    TriggL T3459,vl,laserOFF,z0,toolEtna\WObj:=wobjEtna;
    TriggL T3460,v50,laserON,z0,toolEtna\WObj:=wobjEtna;
    TriggL T3461,vl,laserOFF,z0,toolEtna\WObj:=wobjEtna;
    TriggL T3462,v50,laserON,z0,toolEtna\WObj:=wobjEtna;
    TriggL T3463,vl,laserOFF,z0,toolEtna\WObj:=wobjEtna;
    TriggL T3464,v50,laserON,z0,toolEtna\WObj:=wobjEtna;
    TriggL T3465,vl,laserOFF,z0,toolEtna\WObj:=wobjEtna;
    TriggL T3466,v50,laserON,z0,toolEtna\WObj:=wobjEtna;
    TriggL T3467,vl,laserOFF,z0,toolEtna\WObj:=wobjEtna;
    TriggL T3468,v50,laserON,z0,toolEtna\WObj:=wobjEtna;
    TriggL T3469,vl,laserOFF,z0,toolEtna\WObj:=wobjEtna;
    TriggL T3470,v50,laserON,z0,toolEtna\WObj:=wobjEtna;
    TriggL T3471,vl,laserOFF,z0,toolEtna\WObj:=wobjEtna;
    TriggL T3472,v50,laserON,z0,toolEtna\WObj:=wobjEtna;
    TriggL T3473,vl,laserOFF,z0,toolEtna\WObj:=wobjEtna;
    TriggL T3474,v50,laserON,z0,toolEtna\WObj:=wobjEtna;
    TriggL T3475,vl,laserOFF,z0,toolEtna\WObj:=wobjEtna;
    TriggL T3476,v50,laserON,z0,toolEtna\WObj:=wobjEtna;
    TriggL T3477,vl,laserOFF,z0,toolEtna\WObj:=wobjEtna;
    TriggL T3478,v50,laserON,z0,toolEtna\WObj:=wobjEtna;
    TriggL T3479,vl,laserOFF,z0,toolEtna\WObj:=wobjEtna;
    TriggL T3480,v50,laserON,z0,toolEtna\WObj:=wobjEtna;
    TriggL T3481,vl,laserOFF,z0,toolEtna\WObj:=wobjEtna;
    TriggL T3482,v50,laserON,z0,toolEtna\WObj:=wobjEtna;
    TriggL T3483,vl,laserOFF,z0,toolEtna\WObj:=wobjEtna;
    TriggL T3484,v50,laserON,z0,toolEtna\WObj:=wobjEtna;
    TriggL T3485,vl,laserOFF,z0,toolEtna\WObj:=wobjEtna;
    TriggL T3486,v50,laserON,z0,toolEtna\WObj:=wobjEtna;
    TriggL T3487,vl,laserOFF,z0,toolEtna\WObj:=wobjEtna;
    TriggL T3488,v50,laserON,z0,toolEtna\WObj:=wobjEtna;
    TriggL T3489,vl,laserOFF,z0,toolEtna\WObj:=wobjEtna;
    TriggL T3490,v50,laserON,z0,toolEtna\WObj:=wobjEtna;
    TriggL T3491,vl,laserOFF,z0,toolEtna\WObj:=wobjEtna;
    TriggL T3492,v50,laserON,z0,toolEtna\WObj:=wobjEtna;
    TriggL T3493,vl,laserOFF,z0,toolEtna\WObj:=wobjEtna;
    TriggL T3494,v50,laserON,z0,toolEtna\WObj:=wobjEtna;
    TriggL T3495,vl,laserOFF,z0,toolEtna\WObj:=wobjEtna;
    TriggL T3496,v50,laserON,z0,toolEtna\WObj:=wobjEtna;
    TriggL T3497,vl,laserOFF,z0,toolEtna\WObj:=wobjEtna;
    TriggL T3498,v50,laserON,z0,toolEtna\WObj:=wobjEtna;
    TriggL T3499,vl,laserOFF,z0,toolEtna\WObj:=wobjEtna;
    TriggL T3500,v50,laserON,z0,toolEtna\WObj:=wobjEtna;
    TriggL T3501,vl,laserOFF,z0,toolEtna\WObj:=wobjEtna;
    TriggL T3502,v50,laserON,z0,toolEtna\WObj:=wobjEtna;
    TriggL T3503,vl,laserOFF,z0,toolEtna\WObj:=wobjEtna;
    TriggL T3504,v50,laserON,z0,toolEtna\WObj:=wobjEtna;
    TriggL T3505,vl,laserOFF,z0,toolEtna\WObj:=wobjEtna;
    TriggL T3506,v50,laserON,z0,toolEtna\WObj:=wobjEtna;
    TriggL T3507,vl,laserOFF,z0,toolEtna\WObj:=wobjEtna;
    TriggL T3508,v50,laserON,z0,toolEtna\WObj:=wobjEtna;
    TriggL T3509,vl,laserOFF,z0,toolEtna\WObj:=wobjEtna;
    TriggL T3510,v50,laserON,z0,toolEtna\WObj:=wobjEtna;
    TriggL T3511,vl,laserOFF,z0,toolEtna\WObj:=wobjEtna;
    TriggL T3512,v50,laserON,z0,toolEtna\WObj:=wobjEtna;
    TriggL T3513,vl,laserOFF,z0,toolEtna\WObj:=wobjEtna;
    TriggL T3514,v50,laserON,z0,toolEtna\WObj:=wobjEtna;
    TriggL T3515,vl,laserOFF,z0,toolEtna\WObj:=wobjEtna;
    TriggL T3516,v50,laserON,z0,toolEtna\WObj:=wobjEtna;
    TriggL T3517,vl,laserOFF,z0,toolEtna\WObj:=wobjEtna;
    TriggL T3518,v50,laserON,z0,toolEtna\WObj:=wobjEtna;
    TriggL T3519,vl,laserOFF,z0,toolEtna\WObj:=wobjEtna;
    TriggL T3520,v50,laserON,z0,toolEtna\WObj:=wobjEtna;
    TriggL T3521,vl,laserOFF,z0,toolEtna\WObj:=wobjEtna;
    TriggL T3522,v50,laserON,z0,toolEtna\WObj:=wobjEtna;
    TriggL T3523,vl,laserOFF,z0,toolEtna\WObj:=wobjEtna;
    TriggL T3524,v50,laserON,z0,toolEtna\WObj:=wobjEtna;
    TriggL T3525,vl,laserOFF,z0,toolEtna\WObj:=wobjEtna;
    TriggL T3526,v50,laserON,z0,toolEtna\WObj:=wobjEtna;
    TriggL T3527,vl,laserOFF,z0,toolEtna\WObj:=wobjEtna;
    TriggL T3528,v50,laserON,z0,toolEtna\WObj:=wobjEtna;
    TriggL T3529,vl,laserOFF,z0,toolEtna\WObj:=wobjEtna;
    TriggL T3530,v50,laserON,z0,toolEtna\WObj:=wobjEtna;
    TriggL T3531,vl,laserOFF,z0,toolEtna\WObj:=wobjEtna;
    TriggL T3532,v50,laserON,z0,toolEtna\WObj:=wobjEtna;
    TriggL T3533,vl,laserOFF,z0,toolEtna\WObj:=wobjEtna;
    TriggL T3534,v50,laserON,z0,toolEtna\WObj:=wobjEtna;
    TriggL T3535,vl,laserOFF,z0,toolEtna\WObj:=wobjEtna;
    TriggL T3536,v50,laserON,z0,toolEtna\WObj:=wobjEtna;
    TriggL T3537,vl,laserOFF,z0,toolEtna\WObj:=wobjEtna;
    TriggL T3538,v50,laserON,z0,toolEtna\WObj:=wobjEtna;
    TriggL T3539,vl,laserOFF,z0,toolEtna\WObj:=wobjEtna;
    TriggL T3540,v50,laserON,z0,toolEtna\WObj:=wobjEtna;
    TriggL T3541,vl,laserOFF,z0,toolEtna\WObj:=wobjEtna;
    TriggL T3542,v50,laserON,z0,toolEtna\WObj:=wobjEtna;
    TriggL T3543,vl,laserOFF,z0,toolEtna\WObj:=wobjEtna;
    TriggL T3544,v50,laserON,z0,toolEtna\WObj:=wobjEtna;
    TriggL T3545,vl,laserOFF,z0,toolEtna\WObj:=wobjEtna;
    TriggL T3546,v50,laserON,z0,toolEtna\WObj:=wobjEtna;
    TriggL T3547,vl,laserOFF,z0,toolEtna\WObj:=wobjEtna;
    TriggL T3548,v50,laserON,z0,toolEtna\WObj:=wobjEtna;
    TriggL T3549,vl,laserOFF,z0,toolEtna\WObj:=wobjEtna;
    TriggL T3550,v50,laserON,z0,toolEtna\WObj:=wobjEtna;
    TriggL T3551,vl,laserOFF,z0,toolEtna\WObj:=wobjEtna;
    TriggL T3552,v50,laserON,z0,toolEtna\WObj:=wobjEtna;
    TriggL T3553,vl,laserOFF,z0,toolEtna\WObj:=wobjEtna;
    TriggL T3554,v50,laserON,z0,toolEtna\WObj:=wobjEtna;
    TriggL T3555,vl,laserOFF,z0,toolEtna\WObj:=wobjEtna;
    TriggL T3556,v50,laserON,z0,toolEtna\WObj:=wobjEtna;
    TriggL T3557,vl,laserOFF,z0,toolEtna\WObj:=wobjEtna;
    TriggL T3558,v50,laserON,z0,toolEtna\WObj:=wobjEtna;
    TriggL T3559,vl,laserOFF,z0,toolEtna\WObj:=wobjEtna;
    TriggL T3560,v50,laserON,z0,toolEtna\WObj:=wobjEtna;
    TriggL T3561,vl,laserOFF,z0,toolEtna\WObj:=wobjEtna;
    TriggL T3562,v50,laserON,z0,toolEtna\WObj:=wobjEtna;
    TriggL T3563,vl,laserOFF,z0,toolEtna\WObj:=wobjEtna;
    TriggL T3564,v50,laserON,z0,toolEtna\WObj:=wobjEtna;
    TriggL T3565,vl,laserOFF,z0,toolEtna\WObj:=wobjEtna;
    TriggL T3566,v50,laserON,z0,toolEtna\WObj:=wobjEtna;
    TriggL T3567,vl,laserOFF,z0,toolEtna\WObj:=wobjEtna;
    TriggL T3568,v50,laserON,z0,toolEtna\WObj:=wobjEtna;
    TriggL T3569,vl,laserOFF,z0,toolEtna\WObj:=wobjEtna;
    TriggL T3570,v50,laserON,z0,toolEtna\WObj:=wobjEtna;
    TriggL T3571,vl,laserOFF,z0,toolEtna\WObj:=wobjEtna;
    TriggL T3572,v50,laserON,z0,toolEtna\WObj:=wobjEtna;
    TriggL T3573,vl,laserOFF,z0,toolEtna\WObj:=wobjEtna;
    TriggL T3574,v50,laserON,z0,toolEtna\WObj:=wobjEtna;
    TriggL T3575,vl,laserOFF,z0,toolEtna\WObj:=wobjEtna;
    TriggL T3576,v50,laserON,z0,toolEtna\WObj:=wobjEtna;
    TriggL T3577,vl,laserOFF,z0,toolEtna\WObj:=wobjEtna;
    TriggL T3578,v50,laserON,z0,toolEtna\WObj:=wobjEtna;
    TriggL T3579,vl,laserOFF,z0,toolEtna\WObj:=wobjEtna;
    TriggL T3580,v50,laserON,z0,toolEtna\WObj:=wobjEtna;
    TriggL T3581,vl,laserOFF,z0,toolEtna\WObj:=wobjEtna;
    TriggL T3582,v50,laserON,z0,toolEtna\WObj:=wobjEtna;
    TriggL T3583,vl,laserOFF,z0,toolEtna\WObj:=wobjEtna;
    TriggL T3584,v50,laserON,z0,toolEtna\WObj:=wobjEtna;
    TriggL T3585,vl,laserOFF,z0,toolEtna\WObj:=wobjEtna;
    TriggL T3586,v50,laserON,z0,toolEtna\WObj:=wobjEtna;
    TriggL T3587,vl,laserOFF,z0,toolEtna\WObj:=wobjEtna;
    TriggL T3588,v50,laserON,z0,toolEtna\WObj:=wobjEtna;
    TriggL T3589,vl,laserOFF,z0,toolEtna\WObj:=wobjEtna;
    TriggL T3590,v50,laserON,z0,toolEtna\WObj:=wobjEtna;
    TriggL T3591,vl,laserOFF,z0,toolEtna\WObj:=wobjEtna;
    TriggL T3592,v50,laserON,z0,toolEtna\WObj:=wobjEtna;
    TriggL T3593,vl,laserOFF,z0,toolEtna\WObj:=wobjEtna;
    TriggL T3594,v50,laserON,z0,toolEtna\WObj:=wobjEtna;
    TriggL T3595,vl,laserOFF,z0,toolEtna\WObj:=wobjEtna;
    TriggL T3596,v50,laserON,z0,toolEtna\WObj:=wobjEtna;
    TriggL T3597,vl,laserOFF,z0,toolEtna\WObj:=wobjEtna;
    TriggL T3598,v50,laserON,z0,toolEtna\WObj:=wobjEtna;
    TriggL T3599,vl,laserOFF,z0,toolEtna\WObj:=wobjEtna;
    TriggL T3600,v50,laserON,z0,toolEtna\WObj:=wobjEtna;
    TriggL T3601,vl,laserOFF,z0,toolEtna\WObj:=wobjEtna;
    TriggL T3602,v50,laserON,z0,toolEtna\WObj:=wobjEtna;
    TriggL T3603,vl,laserOFF,z0,toolEtna\WObj:=wobjEtna;
    TriggL T3604,v50,laserON,z0,toolEtna\WObj:=wobjEtna;
    TriggL T3605,vl,laserOFF,z0,toolEtna\WObj:=wobjEtna;
    TriggL T3606,v50,laserON,z0,toolEtna\WObj:=wobjEtna;
    TriggL T3607,vl,laserOFF,z0,toolEtna\WObj:=wobjEtna;
    TriggL T3608,v50,laserON,z0,toolEtna\WObj:=wobjEtna;
    TriggL T3609,vl,laserOFF,z0,toolEtna\WObj:=wobjEtna;
    TriggL T3610,v50,laserON,z0,toolEtna\WObj:=wobjEtna;
    TriggL T3611,vl,laserOFF,z0,toolEtna\WObj:=wobjEtna;
    TriggL T3612,v50,laserON,z0,toolEtna\WObj:=wobjEtna;
    TriggL T3613,vl,laserOFF,z0,toolEtna\WObj:=wobjEtna;
    TriggL T3614,v50,laserON,z0,toolEtna\WObj:=wobjEtna;
    TriggL T3615,vl,laserOFF,z0,toolEtna\WObj:=wobjEtna;
    TriggL T3616,v50,laserON,z0,toolEtna\WObj:=wobjEtna;
    TriggL T3617,vl,laserOFF,z0,toolEtna\WObj:=wobjEtna;
    TriggL T3618,v50,laserON,z0,toolEtna\WObj:=wobjEtna;
    TriggL T3619,vl,laserOFF,z0,toolEtna\WObj:=wobjEtna;
    TriggL T3620,v50,laserON,z0,toolEtna\WObj:=wobjEtna;
    TriggL T3621,vl,laserOFF,z0,toolEtna\WObj:=wobjEtna;
    TriggL T3622,v50,laserON,z0,toolEtna\WObj:=wobjEtna;
    TriggL T3623,vl,laserOFF,z0,toolEtna\WObj:=wobjEtna;
    TriggL T3624,v50,laserON,z0,toolEtna\WObj:=wobjEtna;
    TriggL T3625,vl,laserOFF,z0,toolEtna\WObj:=wobjEtna;
    TriggL T3626,v50,laserON,z0,toolEtna\WObj:=wobjEtna;
    TriggL T3627,vl,laserOFF,z0,toolEtna\WObj:=wobjEtna;
    TriggL T3628,v50,laserON,z0,toolEtna\WObj:=wobjEtna;
    TriggL T3629,vl,laserOFF,z0,toolEtna\WObj:=wobjEtna;
    TriggL T3630,v50,laserON,z0,toolEtna\WObj:=wobjEtna;
    TriggL T3631,vl,laserOFF,z0,toolEtna\WObj:=wobjEtna;
    TriggL T3632,v50,laserON,z0,toolEtna\WObj:=wobjEtna;
    TriggL T3633,vl,laserOFF,z0,toolEtna\WObj:=wobjEtna;
    TriggL T3634,v50,laserON,z0,toolEtna\WObj:=wobjEtna;
    TriggL T3635,vl,laserOFF,z0,toolEtna\WObj:=wobjEtna;
    TriggL T3636,v50,laserON,z0,toolEtna\WObj:=wobjEtna;
    TriggL T3637,vl,laserOFF,z0,toolEtna\WObj:=wobjEtna;
    TriggL T3638,v50,laserON,z0,toolEtna\WObj:=wobjEtna;
    TriggL T3639,vl,laserOFF,z0,toolEtna\WObj:=wobjEtna;
    TriggL T3640,v50,laserON,z0,toolEtna\WObj:=wobjEtna;
    TriggL T3641,vl,laserOFF,z0,toolEtna\WObj:=wobjEtna;
    TriggL T3642,v50,laserON,z0,toolEtna\WObj:=wobjEtna;
    TriggL T3643,vl,laserOFF,z0,toolEtna\WObj:=wobjEtna;
    TriggL T3644,v50,laserON,z0,toolEtna\WObj:=wobjEtna;
    TriggL T3645,vl,laserOFF,z0,toolEtna\WObj:=wobjEtna;
    TriggL T3646,v50,laserON,z0,toolEtna\WObj:=wobjEtna;
    TriggL T3647,vl,laserOFF,z0,toolEtna\WObj:=wobjEtna;
    TriggL T3648,v50,laserON,z0,toolEtna\WObj:=wobjEtna;
    TriggL T3649,vl,laserOFF,z0,toolEtna\WObj:=wobjEtna;
    TriggL T3650,v50,laserON,z0,toolEtna\WObj:=wobjEtna;
    TriggL T3651,vl,laserOFF,z0,toolEtna\WObj:=wobjEtna;
    TriggL T3652,v50,laserON,z0,toolEtna\WObj:=wobjEtna;
    TriggL T3653,vl,laserOFF,z0,toolEtna\WObj:=wobjEtna;
    TriggL T3654,v50,laserON,z0,toolEtna\WObj:=wobjEtna;
    TriggL T3655,vl,laserOFF,z0,toolEtna\WObj:=wobjEtna;
    TriggL T3656,v50,laserON,z0,toolEtna\WObj:=wobjEtna;
    TriggL T3657,vl,laserOFF,z0,toolEtna\WObj:=wobjEtna;
    TriggL T3658,v50,laserON,z0,toolEtna\WObj:=wobjEtna;
    TriggL T3659,vl,laserOFF,z0,toolEtna\WObj:=wobjEtna;
    TriggL T3660,v50,laserON,z0,toolEtna\WObj:=wobjEtna;
    TriggL T3661,vl,laserOFF,z0,toolEtna\WObj:=wobjEtna;
    TriggL T3662,v50,laserON,z0,toolEtna\WObj:=wobjEtna;
    TriggL T3663,vl,laserOFF,z0,toolEtna\WObj:=wobjEtna;
    TriggL T3664,v50,laserON,z0,toolEtna\WObj:=wobjEtna;
    TriggL T3665,vl,laserOFF,z0,toolEtna\WObj:=wobjEtna;
    TriggL T3666,v50,laserON,z0,toolEtna\WObj:=wobjEtna;
    TriggL T3667,vl,laserOFF,z0,toolEtna\WObj:=wobjEtna;
    TriggL T3668,v50,laserON,z0,toolEtna\WObj:=wobjEtna;
    TriggL T3669,vl,laserOFF,z0,toolEtna\WObj:=wobjEtna;
    TriggL T3670,v50,laserON,z0,toolEtna\WObj:=wobjEtna;
    TriggL T3671,vl,laserOFF,z0,toolEtna\WObj:=wobjEtna;
    TriggL T3672,v50,laserON,z0,toolEtna\WObj:=wobjEtna;
    TriggL T3673,vl,laserOFF,z0,toolEtna\WObj:=wobjEtna;
    TriggL T3674,v50,laserON,z0,toolEtna\WObj:=wobjEtna;
    TriggL T3675,vl,laserOFF,z0,toolEtna\WObj:=wobjEtna;
    TriggL T3676,v50,laserON,z0,toolEtna\WObj:=wobjEtna;
    TriggL T3677,vl,laserOFF,z0,toolEtna\WObj:=wobjEtna;
    TriggL T3678,v50,laserON,z0,toolEtna\WObj:=wobjEtna;
    TriggL T3679,vl,laserOFF,z0,toolEtna\WObj:=wobjEtna;
    TriggL T3680,v50,laserON,z0,toolEtna\WObj:=wobjEtna;
    TriggL T3681,vl,laserOFF,z0,toolEtna\WObj:=wobjEtna;
    TriggL T3682,v50,laserON,z0,toolEtna\WObj:=wobjEtna;
    TriggL T3683,vl,laserOFF,z0,toolEtna\WObj:=wobjEtna;
    TriggL T3684,v50,laserON,z0,toolEtna\WObj:=wobjEtna;
    TriggL T3685,vl,laserOFF,z0,toolEtna\WObj:=wobjEtna;
    TriggL T3686,v50,laserON,z0,toolEtna\WObj:=wobjEtna;
    TriggL T3687,vl,laserOFF,z0,toolEtna\WObj:=wobjEtna;
    TriggL T3688,v50,laserON,z0,toolEtna\WObj:=wobjEtna;
    TriggL T3689,vl,laserOFF,z0,toolEtna\WObj:=wobjEtna;
    TriggL T3690,v50,laserON,z0,toolEtna\WObj:=wobjEtna;
    TriggL T3691,vl,laserOFF,z0,toolEtna\WObj:=wobjEtna;
    TriggL T3692,v50,laserON,z0,toolEtna\WObj:=wobjEtna;
    TriggL T3693,vl,laserOFF,z0,toolEtna\WObj:=wobjEtna;
    TriggL T3694,v50,laserON,z0,toolEtna\WObj:=wobjEtna;
    TriggL T3695,vl,laserOFF,z0,toolEtna\WObj:=wobjEtna;
    TriggL T3696,v50,laserON,z0,toolEtna\WObj:=wobjEtna;
    TriggL T3697,vl,laserOFF,z0,toolEtna\WObj:=wobjEtna;
    TriggL T3698,v50,laserON,z0,toolEtna\WObj:=wobjEtna;
    TriggL T3699,vl,laserOFF,z0,toolEtna\WObj:=wobjEtna;
    TriggL T3700,v50,laserON,z0,toolEtna\WObj:=wobjEtna;
    TriggL T3701,vl,laserOFF,z0,toolEtna\WObj:=wobjEtna;
    TriggL T3702,v50,laserON,z0,toolEtna\WObj:=wobjEtna;
    TriggL T3703,vl,laserOFF,z0,toolEtna\WObj:=wobjEtna;
    TriggL T3704,v50,laserON,z0,toolEtna\WObj:=wobjEtna;
    TriggL T3705,vl,laserOFF,z0,toolEtna\WObj:=wobjEtna;
    TriggL T3706,v50,laserON,z0,toolEtna\WObj:=wobjEtna;
    TriggL T3707,vl,laserOFF,z0,toolEtna\WObj:=wobjEtna;
    TriggL T3708,v50,laserON,z0,toolEtna\WObj:=wobjEtna;
    TriggL T3709,vl,laserOFF,z0,toolEtna\WObj:=wobjEtna;
    TriggL T3710,v50,laserON,z0,toolEtna\WObj:=wobjEtna;
    TriggL T3711,vl,laserOFF,z0,toolEtna\WObj:=wobjEtna;
    TriggL T3712,v50,laserON,z0,toolEtna\WObj:=wobjEtna;
    TriggL T3713,vl,laserOFF,z0,toolEtna\WObj:=wobjEtna;
    TriggL T3714,v50,laserON,z0,toolEtna\WObj:=wobjEtna;
    TriggL T3715,vl,laserOFF,z0,toolEtna\WObj:=wobjEtna;
    TriggL T3716,v50,laserON,z0,toolEtna\WObj:=wobjEtna;
    TriggL T3717,vl,laserOFF,z0,toolEtna\WObj:=wobjEtna;
    TriggL T3718,v50,laserON,z0,toolEtna\WObj:=wobjEtna;
    TriggL T3719,vl,laserOFF,z0,toolEtna\WObj:=wobjEtna;
    TriggL T3720,v50,laserON,z0,toolEtna\WObj:=wobjEtna;
    TriggL T3721,vl,laserOFF,z0,toolEtna\WObj:=wobjEtna;
    TriggL T3722,v50,laserON,z0,toolEtna\WObj:=wobjEtna;
    TriggL T3723,vl,laserOFF,z0,toolEtna\WObj:=wobjEtna;
    TriggL T3724,v50,laserON,z0,toolEtna\WObj:=wobjEtna;
    TriggL T3725,vl,laserOFF,z0,toolEtna\WObj:=wobjEtna;
    TriggL T3726,v50,laserON,z0,toolEtna\WObj:=wobjEtna;
    TriggL T3727,vl,laserOFF,z0,toolEtna\WObj:=wobjEtna;
    TriggL T3728,v50,laserON,z0,toolEtna\WObj:=wobjEtna;
    TriggL T3729,vl,laserOFF,z0,toolEtna\WObj:=wobjEtna;
    TriggL T3730,v50,laserON,z0,toolEtna\WObj:=wobjEtna;
    TriggL T3731,vl,laserOFF,z0,toolEtna\WObj:=wobjEtna;
    TriggL T3732,v50,laserON,z0,toolEtna\WObj:=wobjEtna;
    TriggL T3733,vl,laserOFF,z0,toolEtna\WObj:=wobjEtna;
    TriggL T3734,v50,laserON,z0,toolEtna\WObj:=wobjEtna;
    TriggL T3735,vl,laserOFF,z0,toolEtna\WObj:=wobjEtna;
    TriggL T3736,v50,laserON,z0,toolEtna\WObj:=wobjEtna;
    TriggL T3737,vl,laserOFF,z0,toolEtna\WObj:=wobjEtna;
    TriggL T3738,v50,laserON,z0,toolEtna\WObj:=wobjEtna;
    TriggL T3739,vl,laserOFF,z0,toolEtna\WObj:=wobjEtna;
    TriggL T3740,v50,laserON,z0,toolEtna\WObj:=wobjEtna;
    TriggL T3741,vl,laserOFF,z0,toolEtna\WObj:=wobjEtna;
    TriggL T3742,v50,laserON,z0,toolEtna\WObj:=wobjEtna;
    TriggL T3743,vl,laserOFF,z0,toolEtna\WObj:=wobjEtna;
    TriggL T3744,v50,laserON,z0,toolEtna\WObj:=wobjEtna;
    TriggL T3745,vl,laserOFF,z0,toolEtna\WObj:=wobjEtna;
    TriggL T3746,v50,laserON,z0,toolEtna\WObj:=wobjEtna;
    TriggL T3747,vl,laserOFF,z0,toolEtna\WObj:=wobjEtna;
    TriggL T3748,v50,laserON,z0,toolEtna\WObj:=wobjEtna;
    TriggL T3749,vl,laserOFF,z0,toolEtna\WObj:=wobjEtna;
    TriggL T3750,v50,laserON,z0,toolEtna\WObj:=wobjEtna;
    TriggL T3751,vl,laserOFF,z0,toolEtna\WObj:=wobjEtna;
    TriggL T3752,v50,laserON,z0,toolEtna\WObj:=wobjEtna;
    TriggL T3753,vl,laserOFF,z0,toolEtna\WObj:=wobjEtna;
    TriggL T3754,v50,laserON,z0,toolEtna\WObj:=wobjEtna;
    TriggL T3755,vl,laserOFF,z0,toolEtna\WObj:=wobjEtna;
    TriggL T3756,v50,laserON,z0,toolEtna\WObj:=wobjEtna;
    TriggL T3757,vl,laserOFF,z0,toolEtna\WObj:=wobjEtna;
    TriggL T3758,v50,laserON,z0,toolEtna\WObj:=wobjEtna;
    TriggL T3759,vl,laserOFF,z0,toolEtna\WObj:=wobjEtna;
    TriggL T3760,v50,laserON,z0,toolEtna\WObj:=wobjEtna;
    TriggL T3761,vl,laserOFF,z0,toolEtna\WObj:=wobjEtna;
    TriggL T3762,v50,laserON,z0,toolEtna\WObj:=wobjEtna;
    TriggL T3763,vl,laserOFF,z0,toolEtna\WObj:=wobjEtna;
    TriggL T3764,v50,laserON,z0,toolEtna\WObj:=wobjEtna;
    TriggL T3765,vl,laserOFF,z0,toolEtna\WObj:=wobjEtna;
    TriggL T3766,v50,laserON,z0,toolEtna\WObj:=wobjEtna;
    TriggL T3767,vl,laserOFF,z0,toolEtna\WObj:=wobjEtna;
    TriggL T3768,v50,laserON,z0,toolEtna\WObj:=wobjEtna;
    TriggL T3769,vl,laserOFF,z0,toolEtna\WObj:=wobjEtna;
    TriggL T3770,v50,laserON,z0,toolEtna\WObj:=wobjEtna;
    TriggL T3771,vl,laserOFF,z0,toolEtna\WObj:=wobjEtna;
    TriggL T3772,v50,laserON,z0,toolEtna\WObj:=wobjEtna;
    TriggL T3773,vl,laserOFF,z0,toolEtna\WObj:=wobjEtna;
    TriggL T3774,v50,laserON,z0,toolEtna\WObj:=wobjEtna;
    TriggL T3775,vl,laserOFF,z0,toolEtna\WObj:=wobjEtna;
    TriggL T3776,v50,laserON,z0,toolEtna\WObj:=wobjEtna;
    TriggL T3777,vl,laserOFF,z0,toolEtna\WObj:=wobjEtna;
    TriggL T3778,v50,laserON,z0,toolEtna\WObj:=wobjEtna;
    TriggL T3779,vl,laserOFF,z0,toolEtna\WObj:=wobjEtna;
    TriggL T3780,v50,laserON,z0,toolEtna\WObj:=wobjEtna;
    TriggL T3781,vl,laserOFF,z0,toolEtna\WObj:=wobjEtna;
    TriggL T3782,v50,laserON,z0,toolEtna\WObj:=wobjEtna;
    TriggL T3783,vl,laserOFF,z0,toolEtna\WObj:=wobjEtna;
    TriggL T3784,v50,laserON,z0,toolEtna\WObj:=wobjEtna;
    TriggL T3785,vl,laserOFF,z0,toolEtna\WObj:=wobjEtna;
    TriggL T3786,v50,laserON,z0,toolEtna\WObj:=wobjEtna;
    TriggL T3787,vl,laserOFF,z0,toolEtna\WObj:=wobjEtna;
    TriggL T3788,v50,laserON,z0,toolEtna\WObj:=wobjEtna;
    TriggL T3789,vl,laserOFF,z0,toolEtna\WObj:=wobjEtna;
    TriggL T3790,v50,laserON,z0,toolEtna\WObj:=wobjEtna;
    TriggL T3791,vl,laserOFF,z0,toolEtna\WObj:=wobjEtna;
    TriggL T3792,v50,laserON,z0,toolEtna\WObj:=wobjEtna;
    TriggL T3793,vl,laserOFF,z0,toolEtna\WObj:=wobjEtna;
    TriggL T3794,v50,laserON,z0,toolEtna\WObj:=wobjEtna;
    TriggL T3795,vl,laserOFF,z0,toolEtna\WObj:=wobjEtna;
    TriggL T3796,v50,laserON,z0,toolEtna\WObj:=wobjEtna;
    TriggL T3797,vl,laserOFF,z0,toolEtna\WObj:=wobjEtna;
    TriggL T3798,v50,laserON,z0,toolEtna\WObj:=wobjEtna;
    TriggL T3799,vl,laserOFF,z0,toolEtna\WObj:=wobjEtna;
    TriggL T3800,v50,laserON,z0,toolEtna\WObj:=wobjEtna;
    TriggL T3801,vl,laserOFF,z0,toolEtna\WObj:=wobjEtna;
    TriggL T3802,v50,laserON,z0,toolEtna\WObj:=wobjEtna;
    TriggL T3803,vl,laserOFF,z0,toolEtna\WObj:=wobjEtna;
    TriggL T3804,v50,laserON,z0,toolEtna\WObj:=wobjEtna;
    TriggL T3805,vl,laserOFF,z0,toolEtna\WObj:=wobjEtna;
    TriggL T3806,v50,laserON,z0,toolEtna\WObj:=wobjEtna;
    TriggL T3807,vl,laserOFF,z0,toolEtna\WObj:=wobjEtna;
    TriggL T3808,v50,laserON,z0,toolEtna\WObj:=wobjEtna;
    TriggL T3809,vl,laserOFF,z0,toolEtna\WObj:=wobjEtna;
    TriggL T3810,v50,laserON,z0,toolEtna\WObj:=wobjEtna;
    TriggL T3811,vl,laserOFF,z0,toolEtna\WObj:=wobjEtna;
    TriggL T3812,v50,laserON,z0,toolEtna\WObj:=wobjEtna;
    TriggL T3813,vl,laserOFF,z0,toolEtna\WObj:=wobjEtna;
    TriggL T3814,v50,laserON,z0,toolEtna\WObj:=wobjEtna;
    TriggL T3815,vl,laserOFF,z0,toolEtna\WObj:=wobjEtna;
    TriggL T3816,v50,laserON,z0,toolEtna\WObj:=wobjEtna;
    TriggL T3817,vl,laserOFF,z0,toolEtna\WObj:=wobjEtna;
    TriggL T3818,v50,laserON,z0,toolEtna\WObj:=wobjEtna;
    TriggL T3819,vl,laserOFF,z0,toolEtna\WObj:=wobjEtna;
    TriggL T3820,v50,laserON,z0,toolEtna\WObj:=wobjEtna;
    TriggL T3821,vl,laserOFF,z0,toolEtna\WObj:=wobjEtna;
    TriggL T3822,v50,laserON,z0,toolEtna\WObj:=wobjEtna;
    TriggL T3823,vl,laserOFF,z0,toolEtna\WObj:=wobjEtna;
    TriggL T3824,v50,laserON,z0,toolEtna\WObj:=wobjEtna;
    TriggL T3825,vl,laserOFF,z0,toolEtna\WObj:=wobjEtna;
    TriggL T3826,v50,laserON,z0,toolEtna\WObj:=wobjEtna;
    TriggL T3827,vl,laserOFF,z0,toolEtna\WObj:=wobjEtna;
    TriggL T3828,v50,laserON,z0,toolEtna\WObj:=wobjEtna;
    TriggL T3829,vl,laserOFF,z0,toolEtna\WObj:=wobjEtna;
    TriggL T3830,v50,laserON,z0,toolEtna\WObj:=wobjEtna;
    TriggL T3831,vl,laserOFF,z0,toolEtna\WObj:=wobjEtna;
    TriggL T3832,v50,laserON,z0,toolEtna\WObj:=wobjEtna;
    TriggL T3833,vl,laserOFF,z0,toolEtna\WObj:=wobjEtna;
    TriggL T3834,v50,laserON,z0,toolEtna\WObj:=wobjEtna;
    TriggL T3835,vl,laserOFF,z0,toolEtna\WObj:=wobjEtna;
    TriggL T3836,v50,laserON,z0,toolEtna\WObj:=wobjEtna;
    TriggL T3837,vl,laserOFF,z0,toolEtna\WObj:=wobjEtna;
    TriggL T3838,v50,laserON,z0,toolEtna\WObj:=wobjEtna;
    TriggL T3839,vl,laserOFF,z0,toolEtna\WObj:=wobjEtna;
    TriggL T3840,v50,laserON,z0,toolEtna\WObj:=wobjEtna;
    TriggL T3841,vl,laserOFF,z0,toolEtna\WObj:=wobjEtna;
    TriggL T3842,v50,laserON,z0,toolEtna\WObj:=wobjEtna;
    TriggL T3843,vl,laserOFF,z0,toolEtna\WObj:=wobjEtna;
    TriggL T3844,v50,laserON,z0,toolEtna\WObj:=wobjEtna;
    TriggL T3845,vl,laserOFF,z0,toolEtna\WObj:=wobjEtna;
    TriggL T3846,v50,laserON,z0,toolEtna\WObj:=wobjEtna;
    TriggL T3847,vl,laserOFF,z0,toolEtna\WObj:=wobjEtna;
    TriggL T3848,v50,laserON,z0,toolEtna\WObj:=wobjEtna;
    TriggL T3849,vl,laserOFF,z0,toolEtna\WObj:=wobjEtna;
    TriggL T3850,v50,laserON,z0,toolEtna\WObj:=wobjEtna;
    TriggL T3851,vl,laserOFF,z0,toolEtna\WObj:=wobjEtna;
    TriggL T3852,v50,laserON,z0,toolEtna\WObj:=wobjEtna;
    TriggL T3853,vl,laserOFF,z0,toolEtna\WObj:=wobjEtna;
    TriggL T3854,v50,laserON,z0,toolEtna\WObj:=wobjEtna;
    TriggL T3855,vl,laserOFF,z0,toolEtna\WObj:=wobjEtna;
    TriggL T3856,v50,laserON,z0,toolEtna\WObj:=wobjEtna;
    TriggL T3857,vl,laserOFF,z0,toolEtna\WObj:=wobjEtna;
    TriggL T3858,v50,laserON,z0,toolEtna\WObj:=wobjEtna;
    TriggL T3859,vl,laserOFF,z0,toolEtna\WObj:=wobjEtna;
    TriggL T3860,v50,laserON,z0,toolEtna\WObj:=wobjEtna;
    TriggL T3861,vl,laserOFF,z0,toolEtna\WObj:=wobjEtna;
    TriggL T3862,v50,laserON,z0,toolEtna\WObj:=wobjEtna;
    TriggL T3863,vl,laserOFF,z0,toolEtna\WObj:=wobjEtna;
    TriggL T3864,v50,laserON,z0,toolEtna\WObj:=wobjEtna;
    TriggL T3865,vl,laserOFF,z0,toolEtna\WObj:=wobjEtna;
    TriggL T3866,v50,laserON,z0,toolEtna\WObj:=wobjEtna;
    TriggL T3867,vl,laserOFF,z0,toolEtna\WObj:=wobjEtna;
    TriggL T3868,v50,laserON,z0,toolEtna\WObj:=wobjEtna;
    TriggL T3869,vl,laserOFF,z0,toolEtna\WObj:=wobjEtna;
    TriggL T3870,v50,laserON,z0,toolEtna\WObj:=wobjEtna;
    TriggL T3871,vl,laserOFF,z0,toolEtna\WObj:=wobjEtna;
    TriggL T3872,v50,laserON,z0,toolEtna\WObj:=wobjEtna;
    TriggL T3873,vl,laserOFF,z0,toolEtna\WObj:=wobjEtna;
    TriggL T3874,v50,laserON,z0,toolEtna\WObj:=wobjEtna;
    TriggL T3875,vl,laserOFF,z0,toolEtna\WObj:=wobjEtna;
    TriggL T3876,v50,laserON,z0,toolEtna\WObj:=wobjEtna;
    TriggL T3877,vl,laserOFF,z0,toolEtna\WObj:=wobjEtna;
    TriggL T3878,v50,laserON,z0,toolEtna\WObj:=wobjEtna;
    TriggL T3879,vl,laserOFF,z0,toolEtna\WObj:=wobjEtna;
    TriggL T3880,v50,laserON,z0,toolEtna\WObj:=wobjEtna;
    TriggL T3881,vl,laserOFF,z0,toolEtna\WObj:=wobjEtna;
    TriggL T3882,v50,laserON,z0,toolEtna\WObj:=wobjEtna;
    TriggL T3883,vl,laserOFF,z0,toolEtna\WObj:=wobjEtna;
    TriggL T3884,v50,laserON,z0,toolEtna\WObj:=wobjEtna;
    TriggL T3885,vl,laserOFF,z0,toolEtna\WObj:=wobjEtna;
    TriggL T3886,v50,laserON,z0,toolEtna\WObj:=wobjEtna;
    TriggL T3887,vl,laserOFF,z0,toolEtna\WObj:=wobjEtna;
    TriggL T3888,v50,laserON,z0,toolEtna\WObj:=wobjEtna;
    TriggL T3889,vl,laserOFF,z0,toolEtna\WObj:=wobjEtna;
    TriggL T3890,v50,laserON,z0,toolEtna\WObj:=wobjEtna;
    TriggL T3891,vl,laserOFF,z0,toolEtna\WObj:=wobjEtna;
    TriggL T3892,v50,laserON,z0,toolEtna\WObj:=wobjEtna;
    TriggL T3893,vl,laserOFF,z0,toolEtna\WObj:=wobjEtna;
    TriggL T3894,v50,laserON,z0,toolEtna\WObj:=wobjEtna;
    TriggL T3895,vl,laserOFF,z0,toolEtna\WObj:=wobjEtna;
    TriggL T3896,v50,laserON,z0,toolEtna\WObj:=wobjEtna;
    TriggL T3897,vl,laserOFF,z0,toolEtna\WObj:=wobjEtna;
    TriggL T3898,v50,laserON,z0,toolEtna\WObj:=wobjEtna;
    TriggL T3899,vl,laserOFF,z0,toolEtna\WObj:=wobjEtna;
    TriggL T3900,v50,laserON,z0,toolEtna\WObj:=wobjEtna;
    TriggL T3901,vl,laserOFF,z0,toolEtna\WObj:=wobjEtna;
    TriggL T3902,v50,laserON,z0,toolEtna\WObj:=wobjEtna;
    TriggL T3903,vl,laserOFF,z0,toolEtna\WObj:=wobjEtna;
    TriggL T3904,v50,laserON,z0,toolEtna\WObj:=wobjEtna;
    TriggL T3905,vl,laserOFF,z0,toolEtna\WObj:=wobjEtna;
    TriggL T3906,v50,laserON,z0,toolEtna\WObj:=wobjEtna;
    TriggL T3907,vl,laserOFF,z0,toolEtna\WObj:=wobjEtna;
    TriggL T3908,v50,laserON,z0,toolEtna\WObj:=wobjEtna;
    TriggL T3909,vl,laserOFF,z0,toolEtna\WObj:=wobjEtna;
    TriggL T3910,v50,laserON,z0,toolEtna\WObj:=wobjEtna;
    TriggL T3911,vl,laserOFF,z0,toolEtna\WObj:=wobjEtna;
    TriggL T3912,v50,laserON,z0,toolEtna\WObj:=wobjEtna;
    TriggL T3913,vl,laserOFF,z0,toolEtna\WObj:=wobjEtna;
    TriggL T3914,v50,laserON,z0,toolEtna\WObj:=wobjEtna;
    TriggL T3915,vl,laserOFF,z0,toolEtna\WObj:=wobjEtna;
    TriggL T3916,v50,laserON,z0,toolEtna\WObj:=wobjEtna;
    TriggL T3917,vl,laserOFF,z0,toolEtna\WObj:=wobjEtna;
    TriggL T3918,v50,laserON,z0,toolEtna\WObj:=wobjEtna;
    TriggL T3919,vl,laserOFF,z0,toolEtna\WObj:=wobjEtna;
    TriggL T3920,v50,laserON,z0,toolEtna\WObj:=wobjEtna;
    TriggL T3921,vl,laserOFF,z0,toolEtna\WObj:=wobjEtna;
    TriggL T3922,v50,laserON,z0,toolEtna\WObj:=wobjEtna;
    TriggL T3923,vl,laserOFF,z0,toolEtna\WObj:=wobjEtna;
    TriggL T3924,v50,laserON,z0,toolEtna\WObj:=wobjEtna;
    TriggL T3925,vl,laserOFF,z0,toolEtna\WObj:=wobjEtna;
    TriggL T3926,v50,laserON,z0,toolEtna\WObj:=wobjEtna;
    TriggL T3927,vl,laserOFF,z0,toolEtna\WObj:=wobjEtna;
    TriggL T3928,v50,laserON,z0,toolEtna\WObj:=wobjEtna;
    TriggL T3929,vl,laserOFF,z0,toolEtna\WObj:=wobjEtna;
    TriggL T3930,v50,laserON,z0,toolEtna\WObj:=wobjEtna;
    TriggL T3931,vl,laserOFF,z0,toolEtna\WObj:=wobjEtna;
    TriggL T3932,v50,laserON,z0,toolEtna\WObj:=wobjEtna;
    TriggL T3933,vl,laserOFF,z0,toolEtna\WObj:=wobjEtna;
    TriggL T3934,v50,laserON,z0,toolEtna\WObj:=wobjEtna;
    TriggL T3935,vl,laserOFF,z0,toolEtna\WObj:=wobjEtna;
    TriggL T3936,v50,laserON,z0,toolEtna\WObj:=wobjEtna;
    TriggL T3937,vl,laserOFF,z0,toolEtna\WObj:=wobjEtna;
    TriggL T3938,v50,laserON,z0,toolEtna\WObj:=wobjEtna;
    TriggL T3939,vl,laserOFF,z0,toolEtna\WObj:=wobjEtna;
    TriggL T3940,v50,laserON,z0,toolEtna\WObj:=wobjEtna;
    TriggL T3941,vl,laserOFF,z0,toolEtna\WObj:=wobjEtna;
    TriggL T3942,v50,laserON,z0,toolEtna\WObj:=wobjEtna;
    TriggL T3943,vl,laserOFF,z0,toolEtna\WObj:=wobjEtna;
    TriggL T3944,v50,laserON,z0,toolEtna\WObj:=wobjEtna;
    TriggL T3945,vl,laserOFF,z0,toolEtna\WObj:=wobjEtna;
    TriggL T3946,v50,laserON,z0,toolEtna\WObj:=wobjEtna;
    TriggL T3947,vl,laserOFF,z0,toolEtna\WObj:=wobjEtna;
    TriggL T3948,v50,laserON,z0,toolEtna\WObj:=wobjEtna;
    TriggL T3949,vl,laserOFF,z0,toolEtna\WObj:=wobjEtna;
    TriggL T3950,v50,laserON,z0,toolEtna\WObj:=wobjEtna;
    TriggL T3951,vl,laserOFF,z0,toolEtna\WObj:=wobjEtna;
    TriggL T3952,v50,laserON,z0,toolEtna\WObj:=wobjEtna;
    TriggL T3953,vl,laserOFF,z0,toolEtna\WObj:=wobjEtna;
    TriggL T3954,v50,laserON,z0,toolEtna\WObj:=wobjEtna;
    TriggL T3955,vl,laserOFF,z0,toolEtna\WObj:=wobjEtna;
    TriggL T3956,v50,laserON,z0,toolEtna\WObj:=wobjEtna;
    TriggL T3957,vl,laserOFF,z0,toolEtna\WObj:=wobjEtna;
    TriggL T3958,v50,laserON,z0,toolEtna\WObj:=wobjEtna;
    TriggL T3959,vl,laserOFF,z0,toolEtna\WObj:=wobjEtna;
    TriggL T3960,v50,laserON,z0,toolEtna\WObj:=wobjEtna;
    TriggL T3961,vl,laserOFF,z0,toolEtna\WObj:=wobjEtna;
    TriggL T3962,v50,laserON,z0,toolEtna\WObj:=wobjEtna;
    TriggL T3963,vl,laserOFF,z0,toolEtna\WObj:=wobjEtna;
    TriggL T3964,v50,laserON,z0,toolEtna\WObj:=wobjEtna;
    TriggL T3965,vl,laserOFF,z0,toolEtna\WObj:=wobjEtna;
    TriggL T3966,v50,laserON,z0,toolEtna\WObj:=wobjEtna;
    TriggL T3967,vl,laserOFF,z0,toolEtna\WObj:=wobjEtna;
    TriggL T3968,v50,laserON,z0,toolEtna\WObj:=wobjEtna;
    TriggL T3969,vl,laserOFF,z0,toolEtna\WObj:=wobjEtna;
    TriggL T3970,v50,laserON,z0,toolEtna\WObj:=wobjEtna;
    TriggL T3971,vl,laserOFF,z0,toolEtna\WObj:=wobjEtna;
    TriggL T3972,v50,laserON,z0,toolEtna\WObj:=wobjEtna;
    TriggL T3973,vl,laserOFF,z0,toolEtna\WObj:=wobjEtna;
    TriggL T3974,v50,laserON,z0,toolEtna\WObj:=wobjEtna;
    TriggL T3975,vl,laserOFF,z0,toolEtna\WObj:=wobjEtna;
    TriggL T3976,v50,laserON,z0,toolEtna\WObj:=wobjEtna;
    TriggL T3977,vl,laserOFF,z0,toolEtna\WObj:=wobjEtna;
    TriggL T3978,v50,laserON,z0,toolEtna\WObj:=wobjEtna;
    TriggL T3979,vl,laserOFF,z0,toolEtna\WObj:=wobjEtna;
    TriggL T3980,v50,laserON,z0,toolEtna\WObj:=wobjEtna;
    TriggL T3981,vl,laserOFF,z0,toolEtna\WObj:=wobjEtna;
    TriggL T3982,v50,laserON,z0,toolEtna\WObj:=wobjEtna;
    TriggL T3983,vl,laserOFF,z0,toolEtna\WObj:=wobjEtna;
    TriggL T3984,v50,laserON,z0,toolEtna\WObj:=wobjEtna;
    TriggL T3985,vl,laserOFF,z0,toolEtna\WObj:=wobjEtna;
    TriggL T3986,v50,laserON,z0,toolEtna\WObj:=wobjEtna;
    TriggL T3987,vl,laserOFF,z0,toolEtna\WObj:=wobjEtna;
    TriggL T3988,v50,laserON,z0,toolEtna\WObj:=wobjEtna;
    TriggL T3989,vl,laserOFF,z0,toolEtna\WObj:=wobjEtna;
    TriggL T3990,v50,laserON,z0,toolEtna\WObj:=wobjEtna;
    TriggL T3991,vl,laserOFF,z0,toolEtna\WObj:=wobjEtna;
    TriggL T3992,v50,laserON,z0,toolEtna\WObj:=wobjEtna;
    TriggL T3993,vl,laserOFF,z0,toolEtna\WObj:=wobjEtna;
    TriggL T3994,v50,laserON,z0,toolEtna\WObj:=wobjEtna;
    TriggL T3995,vl,laserOFF,z0,toolEtna\WObj:=wobjEtna;
    TriggL T3996,v50,laserON,z0,toolEtna\WObj:=wobjEtna;
    TriggL T3997,vl,laserOFF,z0,toolEtna\WObj:=wobjEtna;
    TriggL T3998,v50,laserON,z0,toolEtna\WObj:=wobjEtna;
    TriggL T3999,vl,laserOFF,z0,toolEtna\WObj:=wobjEtna;
    TriggL T4000,v50,laserON,z0,toolEtna\WObj:=wobjEtna;
    TriggL T4001,vl,laserOFF,z0,toolEtna\WObj:=wobjEtna;
    TriggL T4002,v50,laserON,z0,toolEtna\WObj:=wobjEtna;
    TriggL T4003,vl,laserOFF,z0,toolEtna\WObj:=wobjEtna;
    TriggL T4004,v50,laserON,z0,toolEtna\WObj:=wobjEtna;
    TriggL T4005,vl,laserOFF,z0,toolEtna\WObj:=wobjEtna;
    TriggL T4006,v50,laserON,z0,toolEtna\WObj:=wobjEtna;
    TriggL T4007,vl,laserOFF,z0,toolEtna\WObj:=wobjEtna;
    TriggL T4008,v50,laserON,z0,toolEtna\WObj:=wobjEtna;
    TriggL T4009,vl,laserOFF,z0,toolEtna\WObj:=wobjEtna;
    TriggL T4010,v50,laserON,z0,toolEtna\WObj:=wobjEtna;
    TriggL T4011,vl,laserOFF,z0,toolEtna\WObj:=wobjEtna;
    TriggL T4012,v50,laserON,z0,toolEtna\WObj:=wobjEtna;
    TriggL T4013,vl,laserOFF,z0,toolEtna\WObj:=wobjEtna;
    TriggL T4014,v50,laserON,z0,toolEtna\WObj:=wobjEtna;
    TriggL T4015,vl,laserOFF,z0,toolEtna\WObj:=wobjEtna;
    TriggL T4016,v50,laserON,z0,toolEtna\WObj:=wobjEtna;
    TriggL T4017,vl,laserOFF,z0,toolEtna\WObj:=wobjEtna;
    TriggL T4018,v50,laserON,z0,toolEtna\WObj:=wobjEtna;
    TriggL T4019,vl,laserOFF,z0,toolEtna\WObj:=wobjEtna;
    TriggL T4020,v50,laserON,z0,toolEtna\WObj:=wobjEtna;
    TriggL T4021,vl,laserOFF,z0,toolEtna\WObj:=wobjEtna;
    TriggL T4022,v50,laserON,z0,toolEtna\WObj:=wobjEtna;
    TriggL T4023,vl,laserOFF,z0,toolEtna\WObj:=wobjEtna;
    TriggL T4024,v50,laserON,z0,toolEtna\WObj:=wobjEtna;
    TriggL T4025,vl,laserOFF,z0,toolEtna\WObj:=wobjEtna;
    TriggL T4026,v50,laserON,z0,toolEtna\WObj:=wobjEtna;
    TriggL T4027,vl,laserOFF,z0,toolEtna\WObj:=wobjEtna;
    TriggL T4028,v50,laserON,z0,toolEtna\WObj:=wobjEtna;
    TriggL T4029,vl,laserOFF,z0,toolEtna\WObj:=wobjEtna;
    TriggL T4030,v50,laserON,z0,toolEtna\WObj:=wobjEtna;
    TriggL T4031,vl,laserOFF,z0,toolEtna\WObj:=wobjEtna;
    TriggL T4032,v50,laserON,z0,toolEtna\WObj:=wobjEtna;
    TriggL T4033,vl,laserOFF,z0,toolEtna\WObj:=wobjEtna;
    TriggL T4034,v50,laserON,z0,toolEtna\WObj:=wobjEtna;
    TriggL T4035,vl,laserOFF,z0,toolEtna\WObj:=wobjEtna;
    TriggL T4036,v50,laserON,z0,toolEtna\WObj:=wobjEtna;
    TriggL T4037,vl,laserOFF,z0,toolEtna\WObj:=wobjEtna;
    TriggL T4038,v50,laserON,z0,toolEtna\WObj:=wobjEtna;
    TriggL T4039,vl,laserOFF,z0,toolEtna\WObj:=wobjEtna;
    TriggL T4040,v50,laserON,z0,toolEtna\WObj:=wobjEtna;
    TriggL T4041,vl,laserOFF,z0,toolEtna\WObj:=wobjEtna;
    TriggL T4042,v50,laserON,z0,toolEtna\WObj:=wobjEtna;
    TriggL T4043,vl,laserOFF,z0,toolEtna\WObj:=wobjEtna;
    TriggL T4044,v50,laserON,z0,toolEtna\WObj:=wobjEtna;
    TriggL T4045,vl,laserOFF,z0,toolEtna\WObj:=wobjEtna;
    TriggL T4046,v50,laserON,z0,toolEtna\WObj:=wobjEtna;
    TriggL T4047,vl,laserOFF,z0,toolEtna\WObj:=wobjEtna;
    TriggL T4048,v50,laserON,z0,toolEtna\WObj:=wobjEtna;
    TriggL T4049,vl,laserOFF,z0,toolEtna\WObj:=wobjEtna;
    TriggL T4050,v50,laserON,z0,toolEtna\WObj:=wobjEtna;
    TriggL T4051,vl,laserOFF,z0,toolEtna\WObj:=wobjEtna;
    TriggL T4052,v50,laserON,z0,toolEtna\WObj:=wobjEtna;
    TriggL T4053,vl,laserOFF,z0,toolEtna\WObj:=wobjEtna;
    TriggL T4054,v50,laserON,z0,toolEtna\WObj:=wobjEtna;
    TriggL T4055,vl,laserOFF,z0,toolEtna\WObj:=wobjEtna;
    TriggL T4056,v50,laserON,z0,toolEtna\WObj:=wobjEtna;
    TriggL T4057,vl,laserOFF,z0,toolEtna\WObj:=wobjEtna;
    TriggL T4058,v50,laserON,z0,toolEtna\WObj:=wobjEtna;
    TriggL T4059,vl,laserOFF,z0,toolEtna\WObj:=wobjEtna;
    TriggL T4060,v50,laserON,z0,toolEtna\WObj:=wobjEtna;
    TriggL T4061,vl,laserOFF,z0,toolEtna\WObj:=wobjEtna;
    TriggL T4062,v50,laserON,z0,toolEtna\WObj:=wobjEtna;
    TriggL T4063,vl,laserOFF,z0,toolEtna\WObj:=wobjEtna;
    TriggL T4064,v50,laserON,z0,toolEtna\WObj:=wobjEtna;
    TriggL T4065,vl,laserOFF,z0,toolEtna\WObj:=wobjEtna;
    TriggL T4066,v50,laserON,z0,toolEtna\WObj:=wobjEtna;
    TriggL T4067,vl,laserOFF,z0,toolEtna\WObj:=wobjEtna;
    TriggL T4068,v50,laserON,z0,toolEtna\WObj:=wobjEtna;
    TriggL T4069,vl,laserOFF,z0,toolEtna\WObj:=wobjEtna;
    TriggL T4070,v50,laserON,z0,toolEtna\WObj:=wobjEtna;
    TriggL T4071,vl,laserOFF,z0,toolEtna\WObj:=wobjEtna;
    TriggL T4072,v50,laserON,z0,toolEtna\WObj:=wobjEtna;
    TriggL T4073,vl,laserOFF,z0,toolEtna\WObj:=wobjEtna;
    TriggL T4074,v50,laserON,z0,toolEtna\WObj:=wobjEtna;
    TriggL T4075,vl,laserOFF,z0,toolEtna\WObj:=wobjEtna;
    TriggL T4076,v50,laserON,z0,toolEtna\WObj:=wobjEtna;
    TriggL T4077,vl,laserOFF,z0,toolEtna\WObj:=wobjEtna;
    TriggL T4078,v50,laserON,z0,toolEtna\WObj:=wobjEtna;
    TriggL T4079,vl,laserOFF,z0,toolEtna\WObj:=wobjEtna;
    TriggL T4080,v50,laserON,z0,toolEtna\WObj:=wobjEtna;
    TriggL T4081,vl,laserOFF,z0,toolEtna\WObj:=wobjEtna;
    TriggL T4082,v50,laserON,z0,toolEtna\WObj:=wobjEtna;
    TriggL T4083,vl,laserOFF,z0,toolEtna\WObj:=wobjEtna;
    TriggL T4084,v50,laserON,z0,toolEtna\WObj:=wobjEtna;
    TriggL T4085,vl,laserOFF,z0,toolEtna\WObj:=wobjEtna;
    TriggL T4086,v50,laserON,z0,toolEtna\WObj:=wobjEtna;
    TriggL T4087,vl,laserOFF,z0,toolEtna\WObj:=wobjEtna;
    TriggL T4088,v50,laserON,z0,toolEtna\WObj:=wobjEtna;
    TriggL T4089,vl,laserOFF,z0,toolEtna\WObj:=wobjEtna;
    TriggL T4090,v50,laserON,z0,toolEtna\WObj:=wobjEtna;
    TriggL T4091,vl,laserOFF,z0,toolEtna\WObj:=wobjEtna;
    TriggL T4092,v50,laserON,z0,toolEtna\WObj:=wobjEtna;
    TriggL T4093,vl,laserOFF,z0,toolEtna\WObj:=wobjEtna;
    TriggL T4094,v50,laserON,z0,toolEtna\WObj:=wobjEtna;
    TriggL T4095,vl,laserOFF,z0,toolEtna\WObj:=wobjEtna;
    TriggL T4096,v50,laserON,z0,toolEtna\WObj:=wobjEtna;
    TriggL T4097,vl,laserOFF,z0,toolEtna\WObj:=wobjEtna;
    TriggL T4098,v50,laserON,z0,toolEtna\WObj:=wobjEtna;
    TriggL T4099,vl,laserOFF,z0,toolEtna\WObj:=wobjEtna;
    TriggL T4100,v50,laserON,z0,toolEtna\WObj:=wobjEtna;
    TriggL T4101,vl,laserOFF,z0,toolEtna\WObj:=wobjEtna;
    TriggL T4102,v50,laserON,z0,toolEtna\WObj:=wobjEtna;
    TriggL T4103,vl,laserOFF,z0,toolEtna\WObj:=wobjEtna;
    TriggL T4104,v50,laserON,z0,toolEtna\WObj:=wobjEtna;
    TriggL T4105,vl,laserOFF,z0,toolEtna\WObj:=wobjEtna;
    TriggL T4106,v50,laserON,z0,toolEtna\WObj:=wobjEtna;
    TriggL T4107,vl,laserOFF,z0,toolEtna\WObj:=wobjEtna;
    TriggL T4108,v50,laserON,z0,toolEtna\WObj:=wobjEtna;
    TriggL T4109,vl,laserOFF,z0,toolEtna\WObj:=wobjEtna;
    TriggL T4110,v50,laserON,z0,toolEtna\WObj:=wobjEtna;
    TriggL T4111,vl,laserOFF,z0,toolEtna\WObj:=wobjEtna;
    TriggL T4112,v50,laserON,z0,toolEtna\WObj:=wobjEtna;
    TriggL T4113,vl,laserOFF,z0,toolEtna\WObj:=wobjEtna;
    TriggL T4114,v50,laserON,z0,toolEtna\WObj:=wobjEtna;
    TriggL T4115,vl,laserOFF,z0,toolEtna\WObj:=wobjEtna;
    TriggL T4116,v50,laserON,z0,toolEtna\WObj:=wobjEtna;
    TriggL T4117,vl,laserOFF,z0,toolEtna\WObj:=wobjEtna;
    TriggL T4118,v50,laserON,z0,toolEtna\WObj:=wobjEtna;
    TriggL T4119,vl,laserOFF,z0,toolEtna\WObj:=wobjEtna;
    TriggL T4120,v50,laserON,z0,toolEtna\WObj:=wobjEtna;
    TriggL T4121,vl,laserOFF,z0,toolEtna\WObj:=wobjEtna;
    TriggL T4122,v50,laserON,z0,toolEtna\WObj:=wobjEtna;
    TriggL T4123,vl,laserOFF,z0,toolEtna\WObj:=wobjEtna;
    TriggL T4124,v50,laserON,z0,toolEtna\WObj:=wobjEtna;
    TriggL T4125,vl,laserOFF,z0,toolEtna\WObj:=wobjEtna;
    TriggL T4126,v50,laserON,z0,toolEtna\WObj:=wobjEtna;
    TriggL T4127,vl,laserOFF,z0,toolEtna\WObj:=wobjEtna;
    TriggL T4128,v50,laserON,z0,toolEtna\WObj:=wobjEtna;
    TriggL T4129,vl,laserOFF,z0,toolEtna\WObj:=wobjEtna;
    TriggL T4130,v50,laserON,z0,toolEtna\WObj:=wobjEtna;
    TriggL T4131,vl,laserOFF,z0,toolEtna\WObj:=wobjEtna;
    TriggL T4132,v50,laserON,z0,toolEtna\WObj:=wobjEtna;
    TriggL T4133,vl,laserOFF,z0,toolEtna\WObj:=wobjEtna;
    TriggL T4134,v50,laserON,z0,toolEtna\WObj:=wobjEtna;
    TriggL T4135,vl,laserOFF,z0,toolEtna\WObj:=wobjEtna;
    TriggL T4136,v50,laserON,z0,toolEtna\WObj:=wobjEtna;
    TriggL T4137,vl,laserOFF,z0,toolEtna\WObj:=wobjEtna;
    TriggL T4138,v50,laserON,z0,toolEtna\WObj:=wobjEtna;
    TriggL T4139,vl,laserOFF,z0,toolEtna\WObj:=wobjEtna;
    TriggL T4140,v50,laserON,z0,toolEtna\WObj:=wobjEtna;
    TriggL T4141,vl,laserOFF,z0,toolEtna\WObj:=wobjEtna;
    TriggL T4142,v50,laserON,z0,toolEtna\WObj:=wobjEtna;
    TriggL T4143,vl,laserOFF,z0,toolEtna\WObj:=wobjEtna;
    TriggL T4144,v50,laserON,z0,toolEtna\WObj:=wobjEtna;
    TriggL T4145,vl,laserOFF,z0,toolEtna\WObj:=wobjEtna;
    TriggL T4146,v50,laserON,z0,toolEtna\WObj:=wobjEtna;
    TriggL T4147,vl,laserOFF,z0,toolEtna\WObj:=wobjEtna;
    TriggL T4148,v50,laserON,z0,toolEtna\WObj:=wobjEtna;
    TriggL T4149,vl,laserOFF,z0,toolEtna\WObj:=wobjEtna;
    TriggL T4150,v50,laserON,z0,toolEtna\WObj:=wobjEtna;
    TriggL T4151,vl,laserOFF,z0,toolEtna\WObj:=wobjEtna;
    TriggL T4152,v50,laserON,z0,toolEtna\WObj:=wobjEtna;
    TriggL T4153,vl,laserOFF,z0,toolEtna\WObj:=wobjEtna;
    TriggL T4154,v50,laserON,z0,toolEtna\WObj:=wobjEtna;
    TriggL T4155,vl,laserOFF,z0,toolEtna\WObj:=wobjEtna;
    TriggL T4156,v50,laserON,z0,toolEtna\WObj:=wobjEtna;
    TriggL T4157,vl,laserOFF,z0,toolEtna\WObj:=wobjEtna;
    TriggL T4158,v50,laserON,z0,toolEtna\WObj:=wobjEtna;
    TriggL T4159,vl,laserOFF,z0,toolEtna\WObj:=wobjEtna;
    TriggL T4160,v50,laserON,z0,toolEtna\WObj:=wobjEtna;
    TriggL T4161,vl,laserOFF,z0,toolEtna\WObj:=wobjEtna;
    TriggL T4162,v50,laserON,z0,toolEtna\WObj:=wobjEtna;
    TriggL T4163,vl,laserOFF,z0,toolEtna\WObj:=wobjEtna;
    TriggL T4164,v50,laserON,z0,toolEtna\WObj:=wobjEtna;
    TriggL T4165,vl,laserOFF,z0,toolEtna\WObj:=wobjEtna;
    TriggL T4166,v50,laserON,z0,toolEtna\WObj:=wobjEtna;
    TriggL T4167,vl,laserOFF,z0,toolEtna\WObj:=wobjEtna;
    TriggL T4168,v50,laserON,z0,toolEtna\WObj:=wobjEtna;
    TriggL T4169,vl,laserOFF,z0,toolEtna\WObj:=wobjEtna;
    TriggL T4170,v50,laserON,z0,toolEtna\WObj:=wobjEtna;
    TriggL T4171,vl,laserOFF,z0,toolEtna\WObj:=wobjEtna;
    TriggL T4172,v50,laserON,z0,toolEtna\WObj:=wobjEtna;
    TriggL T4173,vl,laserOFF,z0,toolEtna\WObj:=wobjEtna;
    TriggL T4174,v50,laserON,z0,toolEtna\WObj:=wobjEtna;
    TriggL T4175,vl,laserOFF,z0,toolEtna\WObj:=wobjEtna;
    TriggL T4176,v50,laserON,z0,toolEtna\WObj:=wobjEtna;
    TriggL T4177,vl,laserOFF,z0,toolEtna\WObj:=wobjEtna;
    TriggL T4178,v50,laserON,z0,toolEtna\WObj:=wobjEtna;
    TriggL T4179,vl,laserOFF,z0,toolEtna\WObj:=wobjEtna;
    TriggL T4180,v50,laserON,z0,toolEtna\WObj:=wobjEtna;
    TriggL T4181,vl,laserOFF,z0,toolEtna\WObj:=wobjEtna;
    TriggL T4182,v50,laserON,z0,toolEtna\WObj:=wobjEtna;
    TriggL T4183,vl,laserOFF,z0,toolEtna\WObj:=wobjEtna;
    TriggL T4184,v50,laserON,z0,toolEtna\WObj:=wobjEtna;
    TriggL T4185,vl,laserOFF,z0,toolEtna\WObj:=wobjEtna;
    TriggL T4186,v50,laserON,z0,toolEtna\WObj:=wobjEtna;
    TriggL T4187,vl,laserOFF,z0,toolEtna\WObj:=wobjEtna;
    TriggL T4188,v50,laserON,z0,toolEtna\WObj:=wobjEtna;
    TriggL T4189,vl,laserOFF,z0,toolEtna\WObj:=wobjEtna;
    TriggL T4190,v50,laserON,z0,toolEtna\WObj:=wobjEtna;
    TriggL T4191,vl,laserOFF,z0,toolEtna\WObj:=wobjEtna;
    TriggL T4192,v50,laserON,z0,toolEtna\WObj:=wobjEtna;
    TriggL T4193,vl,laserOFF,z0,toolEtna\WObj:=wobjEtna;
    TriggL T4194,v50,laserON,z0,toolEtna\WObj:=wobjEtna;
    TriggL T4195,vl,laserOFF,z0,toolEtna\WObj:=wobjEtna;
    TriggL T4196,v50,laserON,z0,toolEtna\WObj:=wobjEtna;
    TriggL T4197,vl,laserOFF,z0,toolEtna\WObj:=wobjEtna;
    TriggL T4198,v50,laserON,z0,toolEtna\WObj:=wobjEtna;
    TriggL T4199,vl,laserOFF,z0,toolEtna\WObj:=wobjEtna;
    TriggL T4200,v50,laserON,z0,toolEtna\WObj:=wobjEtna;
    TriggL T4201,vl,laserOFF,z0,toolEtna\WObj:=wobjEtna;
    TriggL T4202,v50,laserON,z0,toolEtna\WObj:=wobjEtna;
    TriggL T4203,vl,laserOFF,z0,toolEtna\WObj:=wobjEtna;
    TriggL T4204,v50,laserON,z0,toolEtna\WObj:=wobjEtna;
    TriggL T4205,vl,laserOFF,z0,toolEtna\WObj:=wobjEtna;
    TriggL T4206,v50,laserON,z0,toolEtna\WObj:=wobjEtna;
    TriggL T4207,vl,laserOFF,z0,toolEtna\WObj:=wobjEtna;
    TriggL T4208,v50,laserON,z0,toolEtna\WObj:=wobjEtna;
    TriggL T4209,vl,laserOFF,z0,toolEtna\WObj:=wobjEtna;
    TriggL T4210,v50,laserON,z0,toolEtna\WObj:=wobjEtna;
    TriggL T4211,vl,laserOFF,z0,toolEtna\WObj:=wobjEtna;
    TriggL T4212,v50,laserON,z0,toolEtna\WObj:=wobjEtna;
    TriggL T4213,vl,laserOFF,z0,toolEtna\WObj:=wobjEtna;
    TriggL T4214,v50,laserON,z0,toolEtna\WObj:=wobjEtna;
    TriggL T4215,vl,laserOFF,z0,toolEtna\WObj:=wobjEtna;
    TriggL T4216,v50,laserON,z0,toolEtna\WObj:=wobjEtna;
    TriggL T4217,vl,laserOFF,z0,toolEtna\WObj:=wobjEtna;
    TriggL T4218,v50,laserON,z0,toolEtna\WObj:=wobjEtna;
    TriggL T4219,vl,laserOFF,z0,toolEtna\WObj:=wobjEtna;
    TriggL T4220,v50,laserON,z0,toolEtna\WObj:=wobjEtna;
    TriggL T4221,vl,laserOFF,z0,toolEtna\WObj:=wobjEtna;
    TriggL T4222,v50,laserON,z0,toolEtna\WObj:=wobjEtna;
    TriggL T4223,vl,laserOFF,z0,toolEtna\WObj:=wobjEtna;
    TriggL T4224,v50,laserON,z0,toolEtna\WObj:=wobjEtna;
    TriggL T4225,vl,laserOFF,z0,toolEtna\WObj:=wobjEtna;
    TriggL T4226,v50,laserON,z0,toolEtna\WObj:=wobjEtna;
    TriggL T4227,vl,laserOFF,z0,toolEtna\WObj:=wobjEtna;
    TriggL T4228,v50,laserON,z0,toolEtna\WObj:=wobjEtna;
    TriggL T4229,vl,laserOFF,z0,toolEtna\WObj:=wobjEtna;
    TriggL T4230,v50,laserON,z0,toolEtna\WObj:=wobjEtna;
    TriggL T4231,vl,laserOFF,z0,toolEtna\WObj:=wobjEtna;
    TriggL T4232,v50,laserON,z0,toolEtna\WObj:=wobjEtna;
    TriggL T4233,vl,laserOFF,z0,toolEtna\WObj:=wobjEtna;
    TriggL T4234,v50,laserON,z0,toolEtna\WObj:=wobjEtna;
    TriggL T4235,vl,laserOFF,z0,toolEtna\WObj:=wobjEtna;
    TriggL T4236,v50,laserON,z0,toolEtna\WObj:=wobjEtna;
    TriggL T4237,vl,laserOFF,z0,toolEtna\WObj:=wobjEtna;
    TriggL T4238,v50,laserON,z0,toolEtna\WObj:=wobjEtna;
    TriggL T4239,vl,laserOFF,z0,toolEtna\WObj:=wobjEtna;
    TriggL T4240,v50,laserON,z0,toolEtna\WObj:=wobjEtna;
    TriggL T4241,vl,laserOFF,z0,toolEtna\WObj:=wobjEtna;
    TriggL T4242,v50,laserON,z0,toolEtna\WObj:=wobjEtna;
    TriggL T4243,vl,laserOFF,z0,toolEtna\WObj:=wobjEtna;
    TriggL T4244,v50,laserON,z0,toolEtna\WObj:=wobjEtna;
    TriggL T4245,vl,laserOFF,z0,toolEtna\WObj:=wobjEtna;
    TriggL T4246,v50,laserON,z0,toolEtna\WObj:=wobjEtna;
    TriggL T4247,vl,laserOFF,z0,toolEtna\WObj:=wobjEtna;
    TriggL T4248,v50,laserON,z0,toolEtna\WObj:=wobjEtna;
    TriggL T4249,vl,laserOFF,z0,toolEtna\WObj:=wobjEtna;
    TriggL T4250,v50,laserON,z0,toolEtna\WObj:=wobjEtna;
    TriggL T4251,vl,laserOFF,z0,toolEtna\WObj:=wobjEtna;
    TriggL T4252,v50,laserON,z0,toolEtna\WObj:=wobjEtna;
    TriggL T4253,vl,laserOFF,z0,toolEtna\WObj:=wobjEtna;
    TriggL T4254,v50,laserON,z0,toolEtna\WObj:=wobjEtna;
    TriggL T4255,vl,laserOFF,z0,toolEtna\WObj:=wobjEtna;
    TriggL T4256,v50,laserON,z0,toolEtna\WObj:=wobjEtna;
    TriggL T4257,vl,laserOFF,z0,toolEtna\WObj:=wobjEtna;
    TriggL T4258,v50,laserON,z0,toolEtna\WObj:=wobjEtna;
    TriggL T4259,vl,laserOFF,z0,toolEtna\WObj:=wobjEtna;
    TriggL T4260,v50,laserON,z0,toolEtna\WObj:=wobjEtna;
    TriggL T4261,vl,laserOFF,z0,toolEtna\WObj:=wobjEtna;
    TriggL T4262,v50,laserON,z0,toolEtna\WObj:=wobjEtna;
    TriggL T4263,vl,laserOFF,z0,toolEtna\WObj:=wobjEtna;
    TriggL T4264,v50,laserON,z0,toolEtna\WObj:=wobjEtna;
    TriggL T4265,vl,laserOFF,z0,toolEtna\WObj:=wobjEtna;
    TriggL T4266,v50,laserON,z0,toolEtna\WObj:=wobjEtna;
    TriggL T4267,vl,laserOFF,z0,toolEtna\WObj:=wobjEtna;
    TriggL T4268,v50,laserON,z0,toolEtna\WObj:=wobjEtna;
    TriggL T4269,vl,laserOFF,z0,toolEtna\WObj:=wobjEtna;
    TriggL T4270,v50,laserON,z0,toolEtna\WObj:=wobjEtna;
    TriggL T4271,vl,laserOFF,z0,toolEtna\WObj:=wobjEtna;
    TriggL T4272,v50,laserON,z0,toolEtna\WObj:=wobjEtna;
    TriggL T4273,vl,laserOFF,z0,toolEtna\WObj:=wobjEtna;
    TriggL T4274,v50,laserON,z0,toolEtna\WObj:=wobjEtna;
    TriggL T4275,vl,laserOFF,z0,toolEtna\WObj:=wobjEtna;
    TriggL T4276,v50,laserON,z0,toolEtna\WObj:=wobjEtna;
    TriggL T4277,vl,laserOFF,z0,toolEtna\WObj:=wobjEtna;
    TriggL T4278,v50,laserON,z0,toolEtna\WObj:=wobjEtna;
    TriggL T4279,vl,laserOFF,z0,toolEtna\WObj:=wobjEtna;
    TriggL T4280,v50,laserON,z0,toolEtna\WObj:=wobjEtna;
    TriggL T4281,vl,laserOFF,z0,toolEtna\WObj:=wobjEtna;
    TriggL T4282,v50,laserON,z0,toolEtna\WObj:=wobjEtna;
    TriggL T4283,vl,laserOFF,z0,toolEtna\WObj:=wobjEtna;
    TriggL T4284,v50,laserON,z0,toolEtna\WObj:=wobjEtna;
    TriggL T4285,vl,laserOFF,z0,toolEtna\WObj:=wobjEtna;
    TriggL T4286,v50,laserON,z0,toolEtna\WObj:=wobjEtna;
    TriggL T4287,vl,laserOFF,z0,toolEtna\WObj:=wobjEtna;
    TriggL T4288,v50,laserON,z0,toolEtna\WObj:=wobjEtna;
    TriggL T4289,vl,laserOFF,z0,toolEtna\WObj:=wobjEtna;
    TriggL T4290,v50,laserON,z0,toolEtna\WObj:=wobjEtna;
    TriggL T4291,vl,laserOFF,z0,toolEtna\WObj:=wobjEtna;
    TriggL T4292,v50,laserON,z0,toolEtna\WObj:=wobjEtna;
    TriggL T4293,vl,laserOFF,z0,toolEtna\WObj:=wobjEtna;
    TriggL T4294,v50,laserON,z0,toolEtna\WObj:=wobjEtna;
    TriggL T4295,vl,laserOFF,z0,toolEtna\WObj:=wobjEtna;
    TriggL T4296,v50,laserON,z0,toolEtna\WObj:=wobjEtna;
    TriggL T4297,vl,laserOFF,z0,toolEtna\WObj:=wobjEtna;
    TriggL T4298,v50,laserON,z0,toolEtna\WObj:=wobjEtna;
    TriggL T4299,vl,laserOFF,z0,toolEtna\WObj:=wobjEtna;
    TriggL T4300,v50,laserON,z0,toolEtna\WObj:=wobjEtna;
    TriggL T4301,vl,laserOFF,z0,toolEtna\WObj:=wobjEtna;
    TriggL T4302,v50,laserON,z0,toolEtna\WObj:=wobjEtna;
    TriggL T4303,vl,laserOFF,z0,toolEtna\WObj:=wobjEtna;
    TriggL T4304,v50,laserON,z0,toolEtna\WObj:=wobjEtna;
    TriggL T4305,vl,laserOFF,z0,toolEtna\WObj:=wobjEtna;
    TriggL T4306,v50,laserON,z0,toolEtna\WObj:=wobjEtna;
    TriggL T4307,vl,laserOFF,z0,toolEtna\WObj:=wobjEtna;
    TriggL T4308,v50,laserON,z0,toolEtna\WObj:=wobjEtna;
    TriggL T4309,vl,laserOFF,z0,toolEtna\WObj:=wobjEtna;
    TriggL T4310,v50,laserON,z0,toolEtna\WObj:=wobjEtna;
    TriggL T4311,vl,laserOFF,z0,toolEtna\WObj:=wobjEtna;
    TriggL T4312,v50,laserON,z0,toolEtna\WObj:=wobjEtna;
    TriggL T4313,vl,laserOFF,z0,toolEtna\WObj:=wobjEtna;
    TriggL T4314,v50,laserON,z0,toolEtna\WObj:=wobjEtna;
    TriggL T4315,vl,laserOFF,z0,toolEtna\WObj:=wobjEtna;
    TriggL T4316,v50,laserON,z0,toolEtna\WObj:=wobjEtna;
    TriggL T4317,vl,laserOFF,z0,toolEtna\WObj:=wobjEtna;
    TriggL T4318,v50,laserON,z0,toolEtna\WObj:=wobjEtna;
    TriggL T4319,vl,laserOFF,z0,toolEtna\WObj:=wobjEtna;
    TriggL T4320,v50,laserON,z0,toolEtna\WObj:=wobjEtna;
    TriggL T4321,vl,laserOFF,z0,toolEtna\WObj:=wobjEtna;
    TriggL T4322,v50,laserON,z0,toolEtna\WObj:=wobjEtna;
    TriggL T4323,vl,laserOFF,z0,toolEtna\WObj:=wobjEtna;
    TriggL T4324,v50,laserON,z0,toolEtna\WObj:=wobjEtna;
    TriggL T4325,vl,laserOFF,z0,toolEtna\WObj:=wobjEtna;
    TriggL T4326,v50,laserON,z0,toolEtna\WObj:=wobjEtna;
    TriggL T4327,vl,laserOFF,z0,toolEtna\WObj:=wobjEtna;
    TriggL T4328,v50,laserON,z0,toolEtna\WObj:=wobjEtna;
    TriggL T4329,vl,laserOFF,z0,toolEtna\WObj:=wobjEtna;
    TriggL T4330,v50,laserON,z0,toolEtna\WObj:=wobjEtna;
    TriggL T4331,vl,laserOFF,z0,toolEtna\WObj:=wobjEtna;
    TriggL T4332,v50,laserON,z0,toolEtna\WObj:=wobjEtna;
    TriggL T4333,vl,laserOFF,z0,toolEtna\WObj:=wobjEtna;
    TriggL T4334,v50,laserON,z0,toolEtna\WObj:=wobjEtna;
    TriggL T4335,vl,laserOFF,z0,toolEtna\WObj:=wobjEtna;
    TriggL T4336,v50,laserON,z0,toolEtna\WObj:=wobjEtna;
    TriggL T4337,vl,laserOFF,z0,toolEtna\WObj:=wobjEtna;
    TriggL T4338,v50,laserON,z0,toolEtna\WObj:=wobjEtna;
    TriggL T4339,vl,laserOFF,z0,toolEtna\WObj:=wobjEtna;
    TriggL T4340,v50,laserON,z0,toolEtna\WObj:=wobjEtna;
    TriggL T4341,vl,laserOFF,z0,toolEtna\WObj:=wobjEtna;
    TriggL T4342,v50,laserON,z0,toolEtna\WObj:=wobjEtna;
    TriggL T4343,vl,laserOFF,z0,toolEtna\WObj:=wobjEtna;
    TriggL T4344,v50,laserON,z0,toolEtna\WObj:=wobjEtna;
    TriggL T4345,vl,laserOFF,z0,toolEtna\WObj:=wobjEtna;
    TriggL T4346,v50,laserON,z0,toolEtna\WObj:=wobjEtna;
    TriggL T4347,vl,laserOFF,z0,toolEtna\WObj:=wobjEtna;
    TriggL T4348,v50,laserON,z0,toolEtna\WObj:=wobjEtna;
    TriggL T4349,vl,laserOFF,z0,toolEtna\WObj:=wobjEtna;
    TriggL T4350,v50,laserON,z0,toolEtna\WObj:=wobjEtna;
    TriggL T4351,vl,laserOFF,z0,toolEtna\WObj:=wobjEtna;
    TriggL T4352,v50,laserON,z0,toolEtna\WObj:=wobjEtna;
    TriggL T4353,vl,laserOFF,z0,toolEtna\WObj:=wobjEtna;
    TriggL T4354,v50,laserON,z0,toolEtna\WObj:=wobjEtna;
    TriggL T4355,vl,laserOFF,z0,toolEtna\WObj:=wobjEtna;
    TriggL T4356,v50,laserON,z0,toolEtna\WObj:=wobjEtna;
    TriggL T4357,vl,laserOFF,z0,toolEtna\WObj:=wobjEtna;
    TriggL T4358,v50,laserON,z0,toolEtna\WObj:=wobjEtna;
    TriggL T4359,vl,laserOFF,z0,toolEtna\WObj:=wobjEtna;
    TriggL T4360,v50,laserON,z0,toolEtna\WObj:=wobjEtna;
    TriggL T4361,vl,laserOFF,z0,toolEtna\WObj:=wobjEtna;
    TriggL T4362,v50,laserON,z0,toolEtna\WObj:=wobjEtna;
    TriggL T4363,vl,laserOFF,z0,toolEtna\WObj:=wobjEtna;
    TriggL T4364,v50,laserON,z0,toolEtna\WObj:=wobjEtna;
    TriggL T4365,vl,laserOFF,z0,toolEtna\WObj:=wobjEtna;
    TriggL T4366,v50,laserON,z0,toolEtna\WObj:=wobjEtna;
    TriggL T4367,vl,laserOFF,z0,toolEtna\WObj:=wobjEtna;
    TriggL T4368,v50,laserON,z0,toolEtna\WObj:=wobjEtna;
    TriggL T4369,vl,laserOFF,z0,toolEtna\WObj:=wobjEtna;
    TriggL T4370,v50,laserON,z0,toolEtna\WObj:=wobjEtna;
    TriggL T4371,vl,laserOFF,z0,toolEtna\WObj:=wobjEtna;
    TriggL T4372,v50,laserON,z0,toolEtna\WObj:=wobjEtna;
    TriggL T4373,vl,laserOFF,z0,toolEtna\WObj:=wobjEtna;
    TriggL T4374,v50,laserON,z0,toolEtna\WObj:=wobjEtna;
    TriggL T4375,vl,laserOFF,z0,toolEtna\WObj:=wobjEtna;
    TriggL T4376,v50,laserON,z0,toolEtna\WObj:=wobjEtna;
    TriggL T4377,vl,laserOFF,z0,toolEtna\WObj:=wobjEtna;
    TriggL T4378,v50,laserON,z0,toolEtna\WObj:=wobjEtna;
    TriggL T4379,vl,laserOFF,z0,toolEtna\WObj:=wobjEtna;
    TriggL T4380,v50,laserON,z0,toolEtna\WObj:=wobjEtna;
    TriggL T4381,vl,laserOFF,z0,toolEtna\WObj:=wobjEtna;
    TriggL T4382,v50,laserON,z0,toolEtna\WObj:=wobjEtna;
    TriggL T4383,vl,laserOFF,z0,toolEtna\WObj:=wobjEtna;
    TriggL T4384,v50,laserON,z0,toolEtna\WObj:=wobjEtna;
    TriggL T4385,vl,laserOFF,z0,toolEtna\WObj:=wobjEtna;
    TriggL T4386,v50,laserON,z0,toolEtna\WObj:=wobjEtna;
    TriggL T4387,vl,laserOFF,z0,toolEtna\WObj:=wobjEtna;
    TriggL T4388,v50,laserON,z0,toolEtna\WObj:=wobjEtna;
    TriggL T4389,vl,laserOFF,z0,toolEtna\WObj:=wobjEtna;
    TriggL T4390,v50,laserON,z0,toolEtna\WObj:=wobjEtna;
    TriggL T4391,vl,laserOFF,z0,toolEtna\WObj:=wobjEtna;
    TriggL T4392,v50,laserON,z0,toolEtna\WObj:=wobjEtna;
    TriggL T4393,vl,laserOFF,z0,toolEtna\WObj:=wobjEtna;
    TriggL T4394,v50,laserON,z0,toolEtna\WObj:=wobjEtna;
    TriggL T4395,vl,laserOFF,z0,toolEtna\WObj:=wobjEtna;
    TriggL T4396,v50,laserON,z0,toolEtna\WObj:=wobjEtna;
    TriggL T4397,vl,laserOFF,z0,toolEtna\WObj:=wobjEtna;
    TriggL T4398,v50,laserON,z0,toolEtna\WObj:=wobjEtna;
    TriggL T4399,vl,laserOFF,z0,toolEtna\WObj:=wobjEtna;
    TriggL T4400,v50,laserON,z0,toolEtna\WObj:=wobjEtna;
    TriggL T4401,vl,laserOFF,z0,toolEtna\WObj:=wobjEtna;
    TriggL T4402,v50,laserON,z0,toolEtna\WObj:=wobjEtna;
    TriggL T4403,vl,laserOFF,z0,toolEtna\WObj:=wobjEtna;
    TriggL T4404,v50,laserON,z0,toolEtna\WObj:=wobjEtna;
    TriggL T4405,vl,laserOFF,z0,toolEtna\WObj:=wobjEtna;
    TriggL T4406,v50,laserON,z0,toolEtna\WObj:=wobjEtna;
    TriggL T4407,vl,laserOFF,z0,toolEtna\WObj:=wobjEtna;
    TriggL T4408,v50,laserON,z0,toolEtna\WObj:=wobjEtna;
    TriggL T4409,vl,laserOFF,z0,toolEtna\WObj:=wobjEtna;
    TriggL T4410,v50,laserON,z0,toolEtna\WObj:=wobjEtna;
    TriggL T4411,vl,laserOFF,z0,toolEtna\WObj:=wobjEtna;
    TriggL T4412,v50,laserON,z0,toolEtna\WObj:=wobjEtna;
    TriggL T4413,vl,laserOFF,z0,toolEtna\WObj:=wobjEtna;
    TriggL T4414,v50,laserON,z0,toolEtna\WObj:=wobjEtna;
    TriggL T4415,vl,laserOFF,z0,toolEtna\WObj:=wobjEtna;
    TriggL T4416,v50,laserON,z0,toolEtna\WObj:=wobjEtna;
    TriggL T4417,vl,laserOFF,z0,toolEtna\WObj:=wobjEtna;
    TriggL T4418,v50,laserON,z0,toolEtna\WObj:=wobjEtna;
    TriggL T4419,vl,laserOFF,z0,toolEtna\WObj:=wobjEtna;
    TriggL T4420,v50,laserON,z0,toolEtna\WObj:=wobjEtna;
    TriggL T4421,vl,laserOFF,z0,toolEtna\WObj:=wobjEtna;
    TriggL T4422,v50,laserON,z0,toolEtna\WObj:=wobjEtna;
    TriggL T4423,vl,laserOFF,z0,toolEtna\WObj:=wobjEtna;
    TriggL T4424,v50,laserON,z0,toolEtna\WObj:=wobjEtna;
    TriggL T4425,vl,laserOFF,z0,toolEtna\WObj:=wobjEtna;
    TriggL T4426,v50,laserON,z0,toolEtna\WObj:=wobjEtna;
    TriggL T4427,vl,laserOFF,z0,toolEtna\WObj:=wobjEtna;
    TriggL T4428,v50,laserON,z0,toolEtna\WObj:=wobjEtna;
    TriggL T4429,vl,laserOFF,z0,toolEtna\WObj:=wobjEtna;
    TriggL T4430,v50,laserON,z0,toolEtna\WObj:=wobjEtna;
    TriggL T4431,vl,laserOFF,z0,toolEtna\WObj:=wobjEtna;
    TriggL T4432,v50,laserON,z0,toolEtna\WObj:=wobjEtna;
    TriggL T4433,vl,laserOFF,z0,toolEtna\WObj:=wobjEtna;
    TriggL T4434,v50,laserON,z0,toolEtna\WObj:=wobjEtna;
    TriggL T4435,vl,laserOFF,z0,toolEtna\WObj:=wobjEtna;
    TriggL T4436,v50,laserON,z0,toolEtna\WObj:=wobjEtna;
    TriggL T4437,vl,laserOFF,z0,toolEtna\WObj:=wobjEtna;
    TriggL T4438,v50,laserON,z0,toolEtna\WObj:=wobjEtna;
    TriggL T4439,vl,laserOFF,z0,toolEtna\WObj:=wobjEtna;
    TriggL T4440,v50,laserON,z0,toolEtna\WObj:=wobjEtna;
    TriggL T4441,vl,laserOFF,z0,toolEtna\WObj:=wobjEtna;
    TriggL T4442,v50,laserON,z0,toolEtna\WObj:=wobjEtna;
    TriggL T4443,vl,laserOFF,z0,toolEtna\WObj:=wobjEtna;
    TriggL T4444,v50,laserON,z0,toolEtna\WObj:=wobjEtna;
    TriggL T4445,vl,laserOFF,z0,toolEtna\WObj:=wobjEtna;
    TriggL T4446,v50,laserON,z0,toolEtna\WObj:=wobjEtna;
    TriggL T4447,vl,laserOFF,z0,toolEtna\WObj:=wobjEtna;
    TriggL T4448,v50,laserON,z0,toolEtna\WObj:=wobjEtna;
    TriggL T4449,vl,laserOFF,z0,toolEtna\WObj:=wobjEtna;
    TriggL T4450,v50,laserON,z0,toolEtna\WObj:=wobjEtna;
    TriggL T4451,vl,laserOFF,z0,toolEtna\WObj:=wobjEtna;
    TriggL T4452,v50,laserON,z0,toolEtna\WObj:=wobjEtna;
    TriggL T4453,vl,laserOFF,z0,toolEtna\WObj:=wobjEtna;
    TriggL T4454,v50,laserON,z0,toolEtna\WObj:=wobjEtna;
    TriggL T4455,vl,laserOFF,z0,toolEtna\WObj:=wobjEtna;
    TriggL T4456,v50,laserON,z0,toolEtna\WObj:=wobjEtna;
    TriggL T4457,vl,laserOFF,z0,toolEtna\WObj:=wobjEtna;
    TriggL T4458,v50,laserON,z0,toolEtna\WObj:=wobjEtna;
    TriggL T4459,vl,laserOFF,z0,toolEtna\WObj:=wobjEtna;
    TriggL T4460,v50,laserON,z0,toolEtna\WObj:=wobjEtna;
    TriggL T4461,vl,laserOFF,z0,toolEtna\WObj:=wobjEtna;
    TriggL T4462,v50,laserON,z0,toolEtna\WObj:=wobjEtna;
    TriggL T4463,vl,laserOFF,z0,toolEtna\WObj:=wobjEtna;
    TriggL T4464,v50,laserON,z0,toolEtna\WObj:=wobjEtna;
    TriggL T4465,vl,laserOFF,z0,toolEtna\WObj:=wobjEtna;
    TriggL T4466,v50,laserON,z0,toolEtna\WObj:=wobjEtna;
    TriggL T4467,vl,laserOFF,z0,toolEtna\WObj:=wobjEtna;
    TriggL T4468,v50,laserON,z0,toolEtna\WObj:=wobjEtna;
    TriggL T4469,vl,laserOFF,z0,toolEtna\WObj:=wobjEtna;
    TriggL T4470,v50,laserON,z0,toolEtna\WObj:=wobjEtna;
    TriggL T4471,vl,laserOFF,z0,toolEtna\WObj:=wobjEtna;
    TriggL T4472,v50,laserON,z0,toolEtna\WObj:=wobjEtna;
    TriggL T4473,vl,laserOFF,z0,toolEtna\WObj:=wobjEtna;
    TriggL T4474,v50,laserON,z0,toolEtna\WObj:=wobjEtna;
    TriggL T4475,vl,laserOFF,z0,toolEtna\WObj:=wobjEtna;
    TriggL T4476,v50,laserON,z0,toolEtna\WObj:=wobjEtna;
    TriggL T4477,vl,laserOFF,z0,toolEtna\WObj:=wobjEtna;
    TriggL T4478,v50,laserON,z0,toolEtna\WObj:=wobjEtna;
    TriggL T4479,vl,laserOFF,z0,toolEtna\WObj:=wobjEtna;
    TriggL T4480,v50,laserON,z0,toolEtna\WObj:=wobjEtna;
    TriggL T4481,vl,laserOFF,z0,toolEtna\WObj:=wobjEtna;
    TriggL T4482,v50,laserON,z0,toolEtna\WObj:=wobjEtna;
    TriggL T4483,vl,laserOFF,z0,toolEtna\WObj:=wobjEtna;
    TriggL T4484,v50,laserON,z0,toolEtna\WObj:=wobjEtna;
    TriggL T4485,vl,laserOFF,z0,toolEtna\WObj:=wobjEtna;
    TriggL T4486,v50,laserON,z0,toolEtna\WObj:=wobjEtna;
    TriggL T4487,vl,laserOFF,z0,toolEtna\WObj:=wobjEtna;
    TriggL T4488,v50,laserON,z0,toolEtna\WObj:=wobjEtna;
    TriggL T4489,vl,laserOFF,z0,toolEtna\WObj:=wobjEtna;
    TriggL T4490,v50,laserON,z0,toolEtna\WObj:=wobjEtna;
    TriggL T4491,vl,laserOFF,z0,toolEtna\WObj:=wobjEtna;
    TriggL T4492,v50,laserON,z0,toolEtna\WObj:=wobjEtna;
    TriggL T4493,vl,laserOFF,z0,toolEtna\WObj:=wobjEtna;
    TriggL T4494,v50,laserON,z0,toolEtna\WObj:=wobjEtna;
    TriggL T4495,vl,laserOFF,z0,toolEtna\WObj:=wobjEtna;
    TriggL T4496,v50,laserON,z0,toolEtna\WObj:=wobjEtna;
    TriggL T4497,vl,laserOFF,z0,toolEtna\WObj:=wobjEtna;
    TriggL T4498,v50,laserON,z0,toolEtna\WObj:=wobjEtna;
    TriggL T4499,vl,laserOFF,z0,toolEtna\WObj:=wobjEtna;
    TriggL T4500,v50,laserON,z0,toolEtna\WObj:=wobjEtna;
    TriggL T4501,vl,laserOFF,z0,toolEtna\WObj:=wobjEtna;
    TriggL T4502,v50,laserON,z0,toolEtna\WObj:=wobjEtna;
    TriggL T4503,vl,laserOFF,z0,toolEtna\WObj:=wobjEtna;
    TriggL T4504,v50,laserON,z0,toolEtna\WObj:=wobjEtna;
    TriggL T4505,vl,laserOFF,z0,toolEtna\WObj:=wobjEtna;
    TriggL T4506,v50,laserON,z0,toolEtna\WObj:=wobjEtna;
    TriggL T4507,vl,laserOFF,z0,toolEtna\WObj:=wobjEtna;
    TriggL T4508,v50,laserON,z0,toolEtna\WObj:=wobjEtna;
    TriggL T4509,vl,laserOFF,z0,toolEtna\WObj:=wobjEtna;
    TriggL T4510,v50,laserON,z0,toolEtna\WObj:=wobjEtna;
    TriggL T4511,vl,laserOFF,z0,toolEtna\WObj:=wobjEtna;
    TriggL T4512,v50,laserON,z0,toolEtna\WObj:=wobjEtna;
    TriggL T4513,vl,laserOFF,z0,toolEtna\WObj:=wobjEtna;
    TriggL T4514,v50,laserON,z0,toolEtna\WObj:=wobjEtna;
    TriggL T4515,vl,laserOFF,z0,toolEtna\WObj:=wobjEtna;
    TriggL T4516,v50,laserON,z0,toolEtna\WObj:=wobjEtna;
    TriggL T4517,vl,laserOFF,z0,toolEtna\WObj:=wobjEtna;
    TriggL T4518,v50,laserON,z0,toolEtna\WObj:=wobjEtna;
    TriggL T4519,vl,laserOFF,z0,toolEtna\WObj:=wobjEtna;
    TriggL T4520,v50,laserON,z0,toolEtna\WObj:=wobjEtna;
    TriggL T4521,vl,laserOFF,z0,toolEtna\WObj:=wobjEtna;
    TriggL T4522,v50,laserON,z0,toolEtna\WObj:=wobjEtna;
    TriggL T4523,vl,laserOFF,z0,toolEtna\WObj:=wobjEtna;
    TriggL T4524,v50,laserON,z0,toolEtna\WObj:=wobjEtna;
    TriggL T4525,vl,laserOFF,z0,toolEtna\WObj:=wobjEtna;
    TriggL T4526,v50,laserON,z0,toolEtna\WObj:=wobjEtna;
    TriggL T4527,vl,laserOFF,z0,toolEtna\WObj:=wobjEtna;
    TriggL T4528,v50,laserON,z0,toolEtna\WObj:=wobjEtna;
    TriggL T4529,vl,laserOFF,z0,toolEtna\WObj:=wobjEtna;
    TriggL T4530,v50,laserON,z0,toolEtna\WObj:=wobjEtna;
    TriggL T4531,vl,laserOFF,z0,toolEtna\WObj:=wobjEtna;
    TriggL T4532,v50,laserON,z0,toolEtna\WObj:=wobjEtna;
    TriggL T4533,vl,laserOFF,z0,toolEtna\WObj:=wobjEtna;
    TriggL T4534,v50,laserON,z0,toolEtna\WObj:=wobjEtna;
    TriggL T4535,vl,laserOFF,z0,toolEtna\WObj:=wobjEtna;
    TriggL T4536,v50,laserON,z0,toolEtna\WObj:=wobjEtna;
    TriggL T4537,vl,laserOFF,z0,toolEtna\WObj:=wobjEtna;
    TriggL T4538,v50,laserON,z0,toolEtna\WObj:=wobjEtna;
    TriggL T4539,vl,laserOFF,z0,toolEtna\WObj:=wobjEtna;
    TriggL T4540,v50,laserON,z0,toolEtna\WObj:=wobjEtna;
    TriggL T4541,vl,laserOFF,z0,toolEtna\WObj:=wobjEtna;
    TriggL T4542,v50,laserON,z0,toolEtna\WObj:=wobjEtna;
    TriggL T4543,vl,laserOFF,z0,toolEtna\WObj:=wobjEtna;
    TriggL T4544,v50,laserON,z0,toolEtna\WObj:=wobjEtna;
    TriggL T4545,vl,laserOFF,z0,toolEtna\WObj:=wobjEtna;
    TriggL T4546,v50,laserON,z0,toolEtna\WObj:=wobjEtna;
    TriggL T4547,vl,laserOFF,z0,toolEtna\WObj:=wobjEtna;
    TriggL T4548,v50,laserON,z0,toolEtna\WObj:=wobjEtna;
    TriggL T4549,vl,laserOFF,z0,toolEtna\WObj:=wobjEtna;
    TriggL T4550,v50,laserON,z0,toolEtna\WObj:=wobjEtna;
    TriggL T4551,vl,laserOFF,z0,toolEtna\WObj:=wobjEtna;
    TriggL T4552,v50,laserON,z0,toolEtna\WObj:=wobjEtna;
    TriggL T4553,vl,laserOFF,z0,toolEtna\WObj:=wobjEtna;
    TriggL T4554,v50,laserON,z0,toolEtna\WObj:=wobjEtna;
    TriggL T4555,vl,laserOFF,z0,toolEtna\WObj:=wobjEtna;
    TriggL T4556,v50,laserON,z0,toolEtna\WObj:=wobjEtna;
    TriggL T4557,vl,laserOFF,z0,toolEtna\WObj:=wobjEtna;
    TriggL T4558,v50,laserON,z0,toolEtna\WObj:=wobjEtna;
    TriggL T4559,vl,laserOFF,z0,toolEtna\WObj:=wobjEtna;
    TriggL T4560,v50,laserON,z0,toolEtna\WObj:=wobjEtna;
    TriggL T4561,vl,laserOFF,z0,toolEtna\WObj:=wobjEtna;
    TriggL T4562,v50,laserON,z0,toolEtna\WObj:=wobjEtna;
    TriggL T4563,vl,laserOFF,z0,toolEtna\WObj:=wobjEtna;
    TriggL T4564,v50,laserON,z0,toolEtna\WObj:=wobjEtna;
    TriggL T4565,vl,laserOFF,z0,toolEtna\WObj:=wobjEtna;
    TriggL T4566,v50,laserON,z0,toolEtna\WObj:=wobjEtna;
    TriggL T4567,vl,laserOFF,z0,toolEtna\WObj:=wobjEtna;
    TriggL T4568,v50,laserON,z0,toolEtna\WObj:=wobjEtna;
    TriggL T4569,vl,laserOFF,z0,toolEtna\WObj:=wobjEtna;
    TriggL T4570,v50,laserON,z0,toolEtna\WObj:=wobjEtna;
    TriggL T4571,vl,laserOFF,z0,toolEtna\WObj:=wobjEtna;
    TriggL T4572,v50,laserON,z0,toolEtna\WObj:=wobjEtna;
    TriggL T4573,vl,laserOFF,z0,toolEtna\WObj:=wobjEtna;
    TriggL T4574,v50,laserON,z0,toolEtna\WObj:=wobjEtna;
    TriggL T4575,vl,laserOFF,z0,toolEtna\WObj:=wobjEtna;
    TriggL T4576,v50,laserON,z0,toolEtna\WObj:=wobjEtna;
    TriggL T4577,vl,laserOFF,z0,toolEtna\WObj:=wobjEtna;
    TriggL T4578,v50,laserON,z0,toolEtna\WObj:=wobjEtna;
    TriggL T4579,vl,laserOFF,z0,toolEtna\WObj:=wobjEtna;
    TriggL T4580,v50,laserON,z0,toolEtna\WObj:=wobjEtna;
    TriggL T4581,vl,laserOFF,z0,toolEtna\WObj:=wobjEtna;
    TriggL T4582,v50,laserON,z0,toolEtna\WObj:=wobjEtna;
    TriggL T4583,vl,laserOFF,z0,toolEtna\WObj:=wobjEtna;
    TriggL T4584,v50,laserON,z0,toolEtna\WObj:=wobjEtna;
    TriggL T4585,vl,laserOFF,z0,toolEtna\WObj:=wobjEtna;
    TriggL T4586,v50,laserON,z0,toolEtna\WObj:=wobjEtna;
    TriggL T4587,vl,laserOFF,z0,toolEtna\WObj:=wobjEtna;
    TriggL T4588,v50,laserON,z0,toolEtna\WObj:=wobjEtna;
    TriggL T4589,vl,laserOFF,z0,toolEtna\WObj:=wobjEtna;
    TriggL T4590,v50,laserON,z0,toolEtna\WObj:=wobjEtna;
    TriggL T4591,vl,laserOFF,z0,toolEtna\WObj:=wobjEtna;
    TriggL T4592,v50,laserON,z0,toolEtna\WObj:=wobjEtna;
    TriggL T4593,vl,laserOFF,z0,toolEtna\WObj:=wobjEtna;
    TriggL T4594,v50,laserON,z0,toolEtna\WObj:=wobjEtna;
    TriggL T4595,vl,laserOFF,z0,toolEtna\WObj:=wobjEtna;
    TriggL T4596,v50,laserON,z0,toolEtna\WObj:=wobjEtna;
    TriggL T4597,vl,laserOFF,z0,toolEtna\WObj:=wobjEtna;
    TriggL T4598,v50,laserON,z0,toolEtna\WObj:=wobjEtna;
    TriggL T4599,vl,laserOFF,z0,toolEtna\WObj:=wobjEtna;
    TriggL T4600,v50,laserON,z0,toolEtna\WObj:=wobjEtna;
    TriggL T4601,vl,laserOFF,z0,toolEtna\WObj:=wobjEtna;
    TriggL T4602,v50,laserON,z0,toolEtna\WObj:=wobjEtna;
    TriggL T4603,vl,laserOFF,z0,toolEtna\WObj:=wobjEtna;
    TriggL T4604,v50,laserON,z0,toolEtna\WObj:=wobjEtna;
    TriggL T4605,vl,laserOFF,z0,toolEtna\WObj:=wobjEtna;
    TriggL T4606,v50,laserON,z0,toolEtna\WObj:=wobjEtna;
    TriggL T4607,vl,laserOFF,z0,toolEtna\WObj:=wobjEtna;
    TriggL T4608,v50,laserON,z0,toolEtna\WObj:=wobjEtna;
    TriggL T4609,vl,laserOFF,z0,toolEtna\WObj:=wobjEtna;
    TriggL T4610,v50,laserON,z0,toolEtna\WObj:=wobjEtna;
    TriggL T4611,vl,laserOFF,z0,toolEtna\WObj:=wobjEtna;
    TriggL T4612,v50,laserON,z0,toolEtna\WObj:=wobjEtna;
    TriggL T4613,vl,laserOFF,z0,toolEtna\WObj:=wobjEtna;
    TriggL T4614,v50,laserON,z0,toolEtna\WObj:=wobjEtna;
    TriggL T4615,vl,laserOFF,z0,toolEtna\WObj:=wobjEtna;
    TriggL T4616,v50,laserON,z0,toolEtna\WObj:=wobjEtna;
    TriggL T4617,vl,laserOFF,z0,toolEtna\WObj:=wobjEtna;
    TriggL T4618,v50,laserON,z0,toolEtna\WObj:=wobjEtna;
    TriggL T4619,vl,laserOFF,z0,toolEtna\WObj:=wobjEtna;
    TriggL T4620,v50,laserON,z0,toolEtna\WObj:=wobjEtna;
    TriggL T4621,vl,laserOFF,z0,toolEtna\WObj:=wobjEtna;
    TriggL T4622,v50,laserON,z0,toolEtna\WObj:=wobjEtna;
    TriggL T4623,vl,laserOFF,z0,toolEtna\WObj:=wobjEtna;
    TriggL T4624,v50,laserON,z0,toolEtna\WObj:=wobjEtna;
    TriggL T4625,vl,laserOFF,z0,toolEtna\WObj:=wobjEtna;
    TriggL T4626,v50,laserON,z0,toolEtna\WObj:=wobjEtna;
    TriggL T4627,vl,laserOFF,z0,toolEtna\WObj:=wobjEtna;
    TriggL T4628,v50,laserON,z0,toolEtna\WObj:=wobjEtna;
    TriggL T4629,vl,laserOFF,z0,toolEtna\WObj:=wobjEtna;
    TriggL T4630,v50,laserON,z0,toolEtna\WObj:=wobjEtna;
    TriggL T4631,vl,laserOFF,z0,toolEtna\WObj:=wobjEtna;
    TriggL T4632,v50,laserON,z0,toolEtna\WObj:=wobjEtna;
    TriggL T4633,vl,laserOFF,z0,toolEtna\WObj:=wobjEtna;
    TriggL T4634,v50,laserON,z0,toolEtna\WObj:=wobjEtna;
    TriggL T4635,vl,laserOFF,z0,toolEtna\WObj:=wobjEtna;
    TriggL T4636,v50,laserON,z0,toolEtna\WObj:=wobjEtna;
    TriggL T4637,vl,laserOFF,z0,toolEtna\WObj:=wobjEtna;
    TriggL T4638,v50,laserON,z0,toolEtna\WObj:=wobjEtna;
    TriggL T4639,vl,laserOFF,z0,toolEtna\WObj:=wobjEtna;
    TriggL T4640,v50,laserON,z0,toolEtna\WObj:=wobjEtna;
    TriggL T4641,vl,laserOFF,z0,toolEtna\WObj:=wobjEtna;
    TriggL T4642,v50,laserON,z0,toolEtna\WObj:=wobjEtna;
    TriggL T4643,vl,laserOFF,z0,toolEtna\WObj:=wobjEtna;
    TriggL T4644,v50,laserON,z0,toolEtna\WObj:=wobjEtna;
    TriggL T4645,vl,laserOFF,z0,toolEtna\WObj:=wobjEtna;
    TriggL T4646,v50,laserON,z0,toolEtna\WObj:=wobjEtna;
    TriggL T4647,vl,laserOFF,z0,toolEtna\WObj:=wobjEtna;
    TriggL T4648,v50,laserON,z0,toolEtna\WObj:=wobjEtna;
    TriggL T4649,vl,laserOFF,z0,toolEtna\WObj:=wobjEtna;
    TriggL T4650,v50,laserON,z0,toolEtna\WObj:=wobjEtna;
    TriggL T4651,vl,laserOFF,z0,toolEtna\WObj:=wobjEtna;
    TriggL T4652,v50,laserON,z0,toolEtna\WObj:=wobjEtna;
    TriggL T4653,vl,laserOFF,z0,toolEtna\WObj:=wobjEtna;
    TriggL T4654,v50,laserON,z0,toolEtna\WObj:=wobjEtna;
    TriggL T4655,vl,laserOFF,z0,toolEtna\WObj:=wobjEtna;
    TriggL T4656,v50,laserON,z0,toolEtna\WObj:=wobjEtna;
    TriggL T4657,vl,laserOFF,z0,toolEtna\WObj:=wobjEtna;
    TriggL T4658,v50,laserON,z0,toolEtna\WObj:=wobjEtna;
    TriggL T4659,vl,laserOFF,z0,toolEtna\WObj:=wobjEtna;
    TriggL T4660,v50,laserON,z0,toolEtna\WObj:=wobjEtna;
    TriggL T4661,vl,laserOFF,z0,toolEtna\WObj:=wobjEtna;
    TriggL T4662,v50,laserON,z0,toolEtna\WObj:=wobjEtna;
    TriggL T4663,vl,laserOFF,z0,toolEtna\WObj:=wobjEtna;
    TriggL T4664,v50,laserON,z0,toolEtna\WObj:=wobjEtna;
    TriggL T4665,vl,laserOFF,z0,toolEtna\WObj:=wobjEtna;
    TriggL T4666,v50,laserON,z0,toolEtna\WObj:=wobjEtna;
    TriggL T4667,vl,laserOFF,z0,toolEtna\WObj:=wobjEtna;
    TriggL T4668,v50,laserON,z0,toolEtna\WObj:=wobjEtna;
    TriggL T4669,vl,laserOFF,z0,toolEtna\WObj:=wobjEtna;
    TriggL T4670,v50,laserON,z0,toolEtna\WObj:=wobjEtna;
    TriggL T4671,vl,laserOFF,z0,toolEtna\WObj:=wobjEtna;
    TriggL T4672,v50,laserON,z0,toolEtna\WObj:=wobjEtna;
    TriggL T4673,vl,laserOFF,z0,toolEtna\WObj:=wobjEtna;
    TriggL T4674,v50,laserON,z0,toolEtna\WObj:=wobjEtna;
    TriggL T4675,vl,laserOFF,z0,toolEtna\WObj:=wobjEtna;
    TriggL T4676,v50,laserON,z0,toolEtna\WObj:=wobjEtna;
    TriggL T4677,vl,laserOFF,z0,toolEtna\WObj:=wobjEtna;
    TriggL T4678,v50,laserON,z0,toolEtna\WObj:=wobjEtna;
    TriggL T4679,vl,laserOFF,z0,toolEtna\WObj:=wobjEtna;
    TriggL T4680,v50,laserON,z0,toolEtna\WObj:=wobjEtna;
    TriggL T4681,vl,laserOFF,z0,toolEtna\WObj:=wobjEtna;
    TriggL T4682,v50,laserON,z0,toolEtna\WObj:=wobjEtna;
    TriggL T4683,vl,laserOFF,z0,toolEtna\WObj:=wobjEtna;
    TriggL T4684,v50,laserON,z0,toolEtna\WObj:=wobjEtna;
    TriggL T4685,vl,laserOFF,z0,toolEtna\WObj:=wobjEtna;
    TriggL T4686,v50,laserON,z0,toolEtna\WObj:=wobjEtna;
    TriggL T4687,vl,laserOFF,z0,toolEtna\WObj:=wobjEtna;
    TriggL T4688,v50,laserON,z0,toolEtna\WObj:=wobjEtna;
    TriggL T4689,vl,laserOFF,z0,toolEtna\WObj:=wobjEtna;
    TriggL T4690,v50,laserON,z0,toolEtna\WObj:=wobjEtna;
    TriggL T4691,vl,laserOFF,z0,toolEtna\WObj:=wobjEtna;
    TriggL T4692,v50,laserON,z0,toolEtna\WObj:=wobjEtna;
    TriggL T4693,vl,laserOFF,z0,toolEtna\WObj:=wobjEtna;
    TriggL T4694,v50,laserON,z0,toolEtna\WObj:=wobjEtna;
    TriggL T4695,vl,laserOFF,z0,toolEtna\WObj:=wobjEtna;
    TriggL T4696,v50,laserON,z0,toolEtna\WObj:=wobjEtna;
    TriggL T4697,vl,laserOFF,z0,toolEtna\WObj:=wobjEtna;
    TriggL T4698,v50,laserON,z0,toolEtna\WObj:=wobjEtna;
    TriggL T4699,vl,laserOFF,z0,toolEtna\WObj:=wobjEtna;
    TriggL T4700,v50,laserON,z0,toolEtna\WObj:=wobjEtna;
    TriggL T4701,vl,laserOFF,z0,toolEtna\WObj:=wobjEtna;
    TriggL T4702,v50,laserON,z0,toolEtna\WObj:=wobjEtna;
    TriggL T4703,vl,laserOFF,z0,toolEtna\WObj:=wobjEtna;
    TriggL T4704,v50,laserON,z0,toolEtna\WObj:=wobjEtna;
    TriggL T4705,vl,laserOFF,z0,toolEtna\WObj:=wobjEtna;
    TriggL T4706,v50,laserON,z0,toolEtna\WObj:=wobjEtna;
    TriggL T4707,vl,laserOFF,z0,toolEtna\WObj:=wobjEtna;
    TriggL T4708,v50,laserON,z0,toolEtna\WObj:=wobjEtna;
    TriggL T4709,vl,laserOFF,z0,toolEtna\WObj:=wobjEtna;
    TriggL T4710,v50,laserON,z0,toolEtna\WObj:=wobjEtna;
    TriggL T4711,vl,laserOFF,z0,toolEtna\WObj:=wobjEtna;
    TriggL T4712,v50,laserON,z0,toolEtna\WObj:=wobjEtna;
    TriggL T4713,vl,laserOFF,z0,toolEtna\WObj:=wobjEtna;
    TriggL T4714,v50,laserON,z0,toolEtna\WObj:=wobjEtna;
    TriggL T4715,vl,laserOFF,z0,toolEtna\WObj:=wobjEtna;
    TriggL T4716,v50,laserON,z0,toolEtna\WObj:=wobjEtna;
    TriggL T4717,vl,laserOFF,z0,toolEtna\WObj:=wobjEtna;
    TriggL T4718,v50,laserON,z0,toolEtna\WObj:=wobjEtna;
    TriggL T4719,vl,laserOFF,z0,toolEtna\WObj:=wobjEtna;
    TriggL T4720,v50,laserON,z0,toolEtna\WObj:=wobjEtna;
    TriggL T4721,vl,laserOFF,z0,toolEtna\WObj:=wobjEtna;
    TriggL T4722,v50,laserON,z0,toolEtna\WObj:=wobjEtna;
    TriggL T4723,vl,laserOFF,z0,toolEtna\WObj:=wobjEtna;
    TriggL T4724,v50,laserON,z0,toolEtna\WObj:=wobjEtna;
    TriggL T4725,vl,laserOFF,z0,toolEtna\WObj:=wobjEtna;
    TriggL T4726,v50,laserON,z0,toolEtna\WObj:=wobjEtna;
    TriggL T4727,vl,laserOFF,z0,toolEtna\WObj:=wobjEtna;
    TriggL T4728,v50,laserON,z0,toolEtna\WObj:=wobjEtna;
    TriggL T4729,vl,laserOFF,z0,toolEtna\WObj:=wobjEtna;
    TriggL T4730,v50,laserON,z0,toolEtna\WObj:=wobjEtna;
    TriggL T4731,vl,laserOFF,z0,toolEtna\WObj:=wobjEtna;
    TriggL T4732,v50,laserON,z0,toolEtna\WObj:=wobjEtna;
    TriggL T4733,vl,laserOFF,z0,toolEtna\WObj:=wobjEtna;

    Reset doLDLStartST;
ENDPROC

PROC mainEtna()
    Set doLDLExtern;
    Set doLDLRequest;
    Set doLDLLaserON;
    WaitDI diLDLLaserON,1;
    Set doLDLStandBy;

    SetGO GoLDL_Prog, 5;
    WaitTime 1;
    SetGO GoLDL_Pwr3, 1200;

    TriggIO laserON, 0\DOp:=doLDLStartST, 1;
    TriggIO laserOFF, 0\DOp:=doLDLStartST, 0;

    Set DoWeldGas;
    !MedicoatL2 "OFF", 5, 20, 7.5;
    MedicoatL1 "OFF", 5, 20, 15;

    MoveJ [[0.0,0.0,100.0],[0.0,0.0,1.0,0.0],[0,0,-1,0],[9E+09,9E+09,9E+09,9E+09,9E+09,9E+09]],v80,z0,toolEtna\WObj:=wobjEtna;

    ConfL \Off;

    cladding;

    MoveJ [[0.0,0.0,100.0],[0.0,0.0,1.0,0.0],[0,0,-1,0],[9E+09,9E+09,9E+09,9E+09,9E+09,9E+09]],v80,z0,toolEtna\WObj:=wobjEtna;

    Reset doMdtPL2On;
    Reset doMdtPL1On;
    Reset DoWeldGas;

    Reset doLDLStandBy;
    Reset doLDLLaserON;
    Reset doLDLRequest;
    Reset doLDLExtern;

ENDPROC

ENDMODULE
